LIN {X 112.363,Y 99.492,Z 63.257,A 180.000,B 0.000,C 180.000} C_DIS
LIN {X 112.396,Y 99.258,Z 63.249,A 180.000,B 0.000,C 180.000} C_DIS
LIN {X 112.406,Y 99.180,Z 63.246,A 180.000,B 0.000,C 180.000} C_DIS
LIN {X 112.413,Y 99.101,Z 63.243,A 180.000,B 0.000,C 180.000} C_DIS
LIN {X 112.420,Y 99.023,Z 63.241,A 180.000,B 0.000,C 180.000} C_DIS
LIN {X 112.433,Y 98.866,Z 63.235,A 180.000,B 0.000,C 180.000} C_DIS
LIN {X 112.453,Y 98.631,Z 63.227,A 180.000,B 0.000,C 180.000} C_DIS
LIN {X 112.466,Y 98.474,Z 63.221,A 180.000,B 0.000,C 180.000} C_DIS
LIN {X 112.473,Y 98.395,Z 63.219,A 180.000,B 0.000,C 180.000} C_DIS
LIN {X 112.478,Y 98.317,Z 63.216,A 180.000,B 0.000,C 180.000} C_DIS
LIN {X 112.480,Y 98.238,Z 63.213,A 180.000,B 0.000,C 180.000} C_DIS
LIN {X 112.494,Y 97.766,Z 63.197,A 180.000,B 0.000,C 180.000} C_DIS
LIN {X 112.498,Y 97.608,Z 63.191,A 180.000,B 0.000,C 180.000} C_DIS
LIN {X 112.500,Y 97.529,Z 63.188,A 180.000,B 0.000,C 180.000} C_DIS
LIN {X 112.500,Y 97.451,Z 63.186,A 180.000,B 0.000,C 180.000} C_DIS
LIN {X 112.497,Y 97.372,Z 63.183,A 180.000,B 0.000,C 180.000} C_DIS
LIN {X 112.493,Y 97.214,Z 63.177,A 180.000,B 0.000,C 180.000} C_DIS
LIN {X 112.491,Y 97.136,Z 63.175,A 180.000,B 0.000,C 180.000} C_DIS
LIN {X 112.486,Y 96.978,Z 63.169,A 180.000,B 0.000,C 180.000} C_DIS
LIN {X 112.480,Y 96.742,Z 63.161,A 180.000,B 0.000,C 180.000} C_DIS
LIN {X 112.477,Y 96.663,Z 63.158,A 180.000,B 0.000,C 180.000} C_DIS
LIN {X 112.471,Y 96.585,Z 63.155,A 180.000,B 0.000,C 180.000} C_DIS
LIN {X 112.458,Y 96.428,Z 63.150,A 180.000,B 0.000,C 180.000} C_DIS
LIN {X 112.418,Y 95.957,Z 63.133,A 180.000,B 0.000,C 180.000} C_DIS
LIN {X 112.412,Y 95.879,Z 63.131,A 180.000,B 0.000,C 180.000} C_DIS
LIN {X 112.403,Y 95.800,Z 63.128,A 180.000,B 0.000,C 180.000} C_DIS
LIN {X 112.393,Y 95.722,Z 63.125,A 180.000,B 0.000,C 180.000} C_DIS
LIN {X 112.305,Y 95.098,Z 63.103,A 180.000,B 0.000,C 180.000} C_DIS
LIN {X 112.293,Y 95.020,Z 63.100,A 180.000,B 0.000,C 180.000} C_DIS
LIN {X 112.280,Y 94.943,Z 63.098,A 180.000,B 0.000,C 180.000} C_DIS
LIN {X 112.265,Y 94.866,Z 63.095,A 180.000,B 0.000,C 180.000} C_DIS
LIN {X 112.142,Y 94.248,Z 63.073,A 180.000,B 0.000,C 180.000} C_DIS
LIN {X 112.126,Y 94.171,Z 63.070,A 180.000,B 0.000,C 180.000} C_DIS
LIN {X 112.107,Y 94.094,Z 63.067,A 180.000,B 0.000,C 180.000} C_DIS
LIN {X 111.989,Y 93.637,Z 63.051,A 180.000,B 0.000,C 180.000} C_DIS
LIN {X 111.930,Y 93.408,Z 63.043,A 180.000,B 0.000,C 180.000} C_DIS
LIN {X 111.909,Y 93.332,Z 63.040,A 180.000,B 0.000,C 180.000} C_DIS
LIN {X 111.886,Y 93.257,Z 63.037,A 180.000,B 0.000,C 180.000} C_DIS
LIN {X 111.695,Y 92.656,Z 63.015,A 180.000,B 0.000,C 180.000} C_DIS
LIN {X 111.670,Y 92.581,Z 63.012,A 180.000,B 0.000,C 180.000} C_DIS
LIN {X 111.644,Y 92.507,Z 63.010,A 180.000,B 0.000,C 180.000} C_DIS
LIN {X 111.616,Y 92.434,Z 63.007,A 180.000,B 0.000,C 180.000} C_DIS
LIN {X 111.392,Y 91.845,Z 62.985,A 180.000,B 0.000,C 180.000} C_DIS
LIN {X 111.363,Y 91.772,Z 62.982,A 180.000,B 0.000,C 180.000} C_DIS
LIN {X 111.332,Y 91.699,Z 62.979,A 180.000,B 0.000,C 180.000} C_DIS
LIN {X 111.203,Y 91.412,Z 62.968,A 180.000,B 0.000,C 180.000} C_DIS
LIN {X 111.043,Y 91.052,Z 62.955,A 180.000,B 0.000,C 180.000} C_DIS
LIN {X 111.009,Y 90.981,Z 62.952,A 180.000,B 0.000,C 180.000} C_DIS
LIN {X 110.974,Y 90.911,Z 62.949,A 180.000,B 0.000,C 180.000} C_DIS
LIN {X 110.685,Y 90.351,Z 62.927,A 180.000,B 0.000,C 180.000} C_DIS
LIN {X 110.648,Y 90.281,Z 62.924,A 180.000,B 0.000,C 180.000} C_DIS
LIN {X 110.610,Y 90.212,Z 62.922,A 180.000,B 0.000,C 180.000} C_DIS
LIN {X 110.570,Y 90.144,Z 62.919,A 180.000,B 0.000,C 180.000} C_DIS
LIN {X 110.250,Y 89.601,Z 62.897,A 180.000,B 0.000,C 180.000} C_DIS
LIN {X 110.210,Y 89.534,Z 62.894,A 180.000,B 0.000,C 180.000} C_DIS
LIN {X 110.167,Y 89.468,Z 62.891,A 180.000,B 0.000,C 180.000} C_DIS
LIN {X 110.124,Y 89.402,Z 62.889,A 180.000,B 0.000,C 180.000} C_DIS
LIN {X 109.992,Y 89.206,Z 62.880,A 180.000,B 0.000,C 180.000} C_DIS
LIN {X 109.905,Y 89.075,Z 62.875,A 180.000,B 0.000,C 180.000} C_DIS
LIN {X 109.774,Y 88.878,Z 62.867,A 180.000,B 0.000,C 180.000} C_DIS
LIN {X 109.729,Y 88.814,Z 62.864,A 180.000,B 0.000,C 180.000} C_DIS
LIN {X 109.682,Y 88.750,Z 62.861,A 180.000,B 0.000,C 180.000} C_DIS
LIN {X 109.351,Y 88.310,Z 62.842,A 180.000,B 0.000,C 180.000} C_DIS
LIN {X 109.303,Y 88.247,Z 62.839,A 180.000,B 0.000,C 180.000} C_DIS
LIN {X 109.256,Y 88.184,Z 62.836,A 180.000,B 0.000,C 180.000} C_DIS
LIN {X 109.207,Y 88.122,Z 62.834,A 180.000,B 0.000,C 180.000} C_DIS
LIN {X 109.156,Y 88.062,Z 62.831,A 180.000,B 0.000,C 180.000} C_DIS
LIN {X 109.055,Y 87.942,Z 62.825,A 180.000,B 0.000,C 180.000} C_DIS
LIN {X 109.004,Y 87.881,Z 62.823,A 180.000,B 0.000,C 180.000} C_DIS
LIN {X 108.902,Y 87.761,Z 62.817,A 180.000,B 0.000,C 180.000} C_DIS
LIN {X 108.750,Y 87.581,Z 62.809,A 180.000,B 0.000,C 180.000} C_DIS
LIN {X 108.699,Y 87.521,Z 62.806,A 180.000,B 0.000,C 180.000} C_DIS
LIN {X 108.646,Y 87.462,Z 62.803,A 180.000,B 0.000,C 180.000} C_DIS
LIN {X 108.592,Y 87.405,Z 62.801,A 180.000,B 0.000,C 180.000} C_DIS
LIN {X 108.483,Y 87.291,Z 62.795,A 180.000,B 0.000,C 180.000} C_DIS
LIN {X 108.159,Y 86.947,Z 62.779,A 180.000,B 0.000,C 180.000} C_DIS
LIN {X 108.104,Y 86.891,Z 62.776,A 180.000,B 0.000,C 180.000} C_DIS
LIN {X 108.047,Y 86.836,Z 62.773,A 180.000,B 0.000,C 180.000} C_DIS
LIN {X 107.876,Y 86.674,Z 62.765,A 180.000,B 0.000,C 180.000} C_DIS
LIN {X 107.761,Y 86.566,Z 62.759,A 180.000,B 0.000,C 180.000} C_DIS
LIN {X 107.704,Y 86.511,Z 62.757,A 180.000,B 0.000,C 180.000} C_DIS
LIN {X 107.590,Y 86.403,Z 62.751,A 180.000,B 0.000,C 180.000} C_DIS
LIN {X 107.532,Y 86.349,Z 62.748,A 180.000,B 0.000,C 180.000} C_DIS
LIN {X 107.474,Y 86.296,Z 62.746,A 180.000,B 0.000,C 180.000} C_DIS
LIN {X 107.414,Y 86.245,Z 62.743,A 180.000,B 0.000,C 180.000} C_DIS
LIN {X 107.294,Y 86.144,Z 62.737,A 180.000,B 0.000,C 180.000} C_DIS
LIN {X 107.233,Y 86.093,Z 62.735,A 180.000,B 0.000,C 180.000} C_DIS
LIN {X 107.113,Y 85.991,Z 62.729,A 180.000,B 0.000,C 180.000} C_DIS
LIN {X 106.933,Y 85.839,Z 62.721,A 180.000,B 0.000,C 180.000} C_DIS
LIN {X 106.872,Y 85.788,Z 62.718,A 180.000,B 0.000,C 180.000} C_DIS
LIN {X 106.810,Y 85.740,Z 62.715,A 180.000,B 0.000,C 180.000} C_DIS
LIN {X 106.747,Y 85.692,Z 62.713,A 180.000,B 0.000,C 180.000} C_DIS
LIN {X 106.622,Y 85.598,Z 62.707,A 180.000,B 0.000,C 180.000} C_DIS
LIN {X 106.433,Y 85.456,Z 62.699,A 180.000,B 0.000,C 180.000} C_DIS
LIN {X 106.307,Y 85.361,Z 62.693,A 180.000,B 0.000,C 180.000} C_DIS
LIN {X 106.244,Y 85.313,Z 62.691,A 180.000,B 0.000,C 180.000} C_DIS
LIN {X 106.180,Y 85.267,Z 62.688,A 180.000,B 0.000,C 180.000} C_DIS
LIN {X 106.116,Y 85.222,Z 62.685,A 180.000,B 0.000,C 180.000} C_DIS
LIN {X 105.985,Y 85.135,Z 62.680,A 180.000,B 0.000,C 180.000} C_DIS
LIN {X 105.854,Y 85.047,Z 62.674,A 180.000,B 0.000,C 180.000} C_DIS
LIN {X 105.723,Y 84.960,Z 62.669,A 180.000,B 0.000,C 180.000} C_DIS
LIN {X 105.592,Y 84.872,Z 62.664,A 180.000,B 0.000,C 180.000} C_DIS
LIN {X 105.526,Y 84.829,Z 62.661,A 180.000,B 0.000,C 180.000} C_DIS
LIN {X 105.460,Y 84.786,Z 62.659,A 180.000,B 0.000,C 180.000} C_DIS
LIN {X 105.392,Y 84.746,Z 62.656,A 180.000,B 0.000,C 180.000} C_DIS
LIN {X 105.324,Y 84.706,Z 62.654,A 180.000,B 0.000,C 180.000} C_DIS
LIN {X 105.257,Y 84.666,Z 62.651,A 180.000,B 0.000,C 180.000} C_DIS
LIN {X 105.189,Y 84.626,Z 62.649,A 180.000,B 0.000,C 180.000} C_DIS
LIN {X 105.053,Y 84.546,Z 62.644,A 180.000,B 0.000,C 180.000} C_DIS
LIN {X 104.917,Y 84.466,Z 62.639,A 180.000,B 0.000,C 180.000} C_DIS
LIN {X 104.782,Y 84.386,Z 62.634,A 180.000,B 0.000,C 180.000} C_DIS
LIN {X 104.643,Y 84.312,Z 62.629,A 180.000,B 0.000,C 180.000} C_DIS
LIN {X 104.503,Y 84.240,Z 62.624,A 180.000,B 0.000,C 180.000} C_DIS
LIN {X 104.363,Y 84.167,Z 62.620,A 180.000,B 0.000,C 180.000} C_DIS
LIN {X 104.223,Y 84.095,Z 62.615,A 180.000,B 0.000,C 180.000} C_DIS
LIN {X 104.083,Y 84.023,Z 62.610,A 180.000,B 0.000,C 180.000} C_DIS
LIN {X 103.941,Y 83.954,Z 62.606,A 180.000,B 0.000,C 180.000} C_DIS
LIN {X 103.797,Y 83.890,Z 62.602,A 180.000,B 0.000,C 180.000} C_DIS
LIN {X 103.654,Y 83.826,Z 62.597,A 180.000,B 0.000,C 180.000} C_DIS
LIN {X 103.510,Y 83.761,Z 62.593,A 180.000,B 0.000,C 180.000} C_DIS
LIN {X 103.366,Y 83.697,Z 62.589,A 180.000,B 0.000,C 180.000} C_DIS
LIN {X 103.222,Y 83.634,Z 62.585,A 180.000,B 0.000,C 180.000} C_DIS
LIN {X 103.075,Y 83.578,Z 62.581,A 180.000,B 0.000,C 180.000} C_DIS
LIN {X 102.927,Y 83.521,Z 62.577,A 180.000,B 0.000,C 180.000} C_DIS
LIN {X 102.780,Y 83.465,Z 62.573,A 180.000,B 0.000,C 180.000} C_DIS
LIN {X 102.633,Y 83.409,Z 62.570,A 180.000,B 0.000,C 180.000} C_DIS
LIN {X 102.486,Y 83.353,Z 62.566,A 180.000,B 0.000,C 180.000} C_DIS
LIN {X 102.337,Y 83.303,Z 62.562,A 180.000,B 0.000,C 180.000} C_DIS
LIN {X 102.186,Y 83.255,Z 62.559,A 180.000,B 0.000,C 180.000} C_DIS
LIN {X 102.036,Y 83.208,Z 62.556,A 180.000,B 0.000,C 180.000} C_DIS
LIN {X 101.886,Y 83.160,Z 62.552,A 180.000,B 0.000,C 180.000} C_DIS
LIN {X 101.736,Y 83.112,Z 62.549,A 180.000,B 0.000,C 180.000} C_DIS
LIN {X 101.585,Y 83.068,Z 62.546,A 180.000,B 0.000,C 180.000} C_DIS
LIN {X 101.433,Y 83.028,Z 62.543,A 180.000,B 0.000,C 180.000} C_DIS
LIN {X 101.280,Y 82.989,Z 62.540,A 180.000,B 0.000,C 180.000} C_DIS
LIN {X 101.128,Y 82.950,Z 62.537,A 180.000,B 0.000,C 180.000} C_DIS
LIN {X 100.975,Y 82.910,Z 62.534,A 180.000,B 0.000,C 180.000} C_DIS
LIN {X 100.822,Y 82.873,Z 62.532,A 180.000,B 0.000,C 180.000} C_DIS
LIN {X 100.668,Y 82.841,Z 62.529,A 180.000,B 0.000,C 180.000} C_DIS
LIN {X 100.513,Y 82.811,Z 62.527,A 180.000,B 0.000,C 180.000} C_DIS
LIN {X 100.204,Y 82.749,Z 62.522,A 180.000,B 0.000,C 180.000} C_DIS
LIN {X 99.894,Y 82.694,Z 62.518,A 180.000,B 0.000,C 180.000} C_DIS
LIN {X 99.582,Y 82.650,Z 62.514,A 180.000,B 0.000,C 180.000} C_DIS
LIN {X 99.270,Y 82.606,Z 62.511,A 180.000,B 0.000,C 180.000} C_DIS
LIN {X 98.957,Y 82.575,Z 62.508,A 180.000,B 0.000,C 180.000} C_DIS
LIN {X 98.643,Y 82.548,Z 62.505,A 180.000,B 0.000,C 180.000} C_DIS
LIN {X 98.329,Y 82.523,Z 62.503,A 180.000,B 0.000,C 180.000} C_DIS
LIN {X 98.014,Y 82.513,Z 62.502,A 180.000,B 0.000,C 180.000} C_DIS
LIN {X 97.699,Y 82.505,Z 62.501,A 180.000,B 0.000,C 180.000} C_DIS
LIN {X 97.385,Y 82.502,Z 62.500,A 180.000,B 0.000,C 180.000} C_DIS
LIN {X 97.153,Y 82.509,Z 62.500,A 180.000,B 0.000,C 180.000} C_DIS
; Cutting Move Starts
LIN {X 96.897,Y 82.516,Z 62.500,A 180.000,B 0.000,C 180.000} C_DIS
LIN {X 96.718,Y 82.521,Z 62.500,A 180.000,B 0.000,C 180.000} C_DIS
LIN {X 96.539,Y 82.533,Z 62.500,A 180.000,B 0.000,C 180.000} C_DIS
LIN {X 96.003,Y 82.578,Z 62.500,A 180.000,B 0.000,C 180.000} C_DIS
LIN {X 95.824,Y 82.594,Z 62.500,A 180.000,B 0.000,C 180.000} C_DIS
LIN {X 95.815,Y 82.595,Z 62.500,A 180.000,B 0.000,C 180.000} C_DIS
LIN {X 95.645,Y 82.618,Z 62.500,A 180.000,B 0.000,C 180.000} C_DIS
LIN {X 95.109,Y 82.694,Z 62.500,A 180.000,B 0.000,C 180.000} C_DIS
LIN {X 94.930,Y 82.722,Z 62.500,A 180.000,B 0.000,C 180.000} C_DIS
LIN {X 94.751,Y 82.758,Z 62.500,A 180.000,B 0.000,C 180.000} C_DIS
LIN {X 94.394,Y 82.829,Z 62.500,A 180.000,B 0.000,C 180.000} C_DIS
LIN {X 94.215,Y 82.865,Z 62.500,A 180.000,B 0.000,C 180.000} C_DIS
LIN {X 94.036,Y 82.908,Z 62.500,A 180.000,B 0.000,C 180.000} C_DIS
LIN {X 93.500,Y 83.046,Z 62.500,A 180.000,B 0.000,C 180.000} C_DIS
LIN {X 93.321,Y 83.094,Z 62.500,A 180.000,B 0.000,C 180.000} C_DIS
LIN {X 93.203,Y 83.131,Z 62.500,A 180.000,B 0.000,C 180.000} C_DIS
LIN {X 92.642,Y 83.310,Z 62.500,A 180.000,B 0.000,C 180.000} C_DIS
LIN {X 92.606,Y 83.322,Z 62.500,A 180.000,B 0.000,C 180.000} C_DIS
LIN {X 92.427,Y 83.386,Z 62.500,A 180.000,B 0.000,C 180.000} C_DIS
LIN {X 91.891,Y 83.591,Z 62.500,A 180.000,B 0.000,C 180.000} C_DIS
LIN {X 91.712,Y 83.662,Z 62.500,A 180.000,B 0.000,C 180.000} C_DIS
LIN {X 91.700,Y 83.668,Z 62.500,A 180.000,B 0.000,C 180.000} C_DIS
LIN {X 91.176,Y 83.902,Z 62.500,A 180.000,B 0.000,C 180.000} C_DIS
LIN {X 90.997,Y 83.983,Z 62.500,A 180.000,B 0.000,C 180.000} C_DIS
LIN {X 90.913,Y 84.025,Z 62.500,A 180.000,B 0.000,C 180.000} C_DIS
LIN {X 90.461,Y 84.259,Z 62.500,A 180.000,B 0.000,C 180.000} C_DIS
LIN {X 90.282,Y 84.351,Z 62.500,A 180.000,B 0.000,C 180.000} C_DIS
LIN {X 90.225,Y 84.383,Z 62.500,A 180.000,B 0.000,C 180.000} C_DIS
LIN {X 90.103,Y 84.454,Z 62.500,A 180.000,B 0.000,C 180.000} C_DIS
LIN {X 89.618,Y 84.740,Z 62.500,A 180.000,B 0.000,C 180.000} C_DIS
LIN {X 89.567,Y 84.770,Z 62.500,A 180.000,B 0.000,C 180.000} C_DIS
LIN {X 89.388,Y 84.886,Z 62.500,A 180.000,B 0.000,C 180.000} C_DIS
LIN {X 89.031,Y 85.125,Z 62.500,A 180.000,B 0.000,C 180.000} C_DIS
LIN {X 88.852,Y 85.244,Z 62.500,A 180.000,B 0.000,C 180.000} C_DIS
LIN {X 88.806,Y 85.276,Z 62.500,A 180.000,B 0.000,C 180.000} C_DIS
LIN {X 88.673,Y 85.376,Z 62.500,A 180.000,B 0.000,C 180.000} C_DIS
LIN {X 88.316,Y 85.645,Z 62.500,A 180.000,B 0.000,C 180.000} C_DIS
LIN {X 88.137,Y 85.781,Z 62.500,A 180.000,B 0.000,C 180.000} C_DIS
LIN {X 88.098,Y 85.813,Z 62.500,A 180.000,B 0.000,C 180.000} C_DIS
LIN {X 87.779,Y 86.082,Z 62.500,A 180.000,B 0.000,C 180.000} C_DIS
LIN {X 87.601,Y 86.233,Z 62.500,A 180.000,B 0.000,C 180.000} C_DIS
LIN {X 87.468,Y 86.349,Z 62.500,A 180.000,B 0.000,C 180.000} C_DIS
LIN {X 87.422,Y 86.393,Z 62.500,A 180.000,B 0.000,C 180.000} C_DIS
LIN {X 87.064,Y 86.731,Z 62.500,A 180.000,B 0.000,C 180.000} C_DIS
LIN {X 86.901,Y 86.885,Z 62.500,A 180.000,B 0.000,C 180.000} C_DIS
LIN {X 86.885,Y 86.901,Z 62.500,A 180.000,B 0.000,C 180.000} C_DIS
LIN {X 86.731,Y 87.064,Z 62.500,A 180.000,B 0.000,C 180.000} C_DIS
LIN {X 86.393,Y 87.422,Z 62.500,A 180.000,B 0.000,C 180.000} C_DIS
LIN {X 86.349,Y 87.468,Z 62.500,A 180.000,B 0.000,C 180.000} C_DIS
LIN {X 86.233,Y 87.601,Z 62.500,A 180.000,B 0.000,C 180.000} C_DIS
LIN {X 85.931,Y 87.958,Z 62.500,A 180.000,B 0.000,C 180.000} C_DIS
LIN {X 85.813,Y 88.098,Z 62.500,A 180.000,B 0.000,C 180.000} C_DIS
LIN {X 85.781,Y 88.137,Z 62.500,A 180.000,B 0.000,C 180.000} C_DIS
LIN {X 85.645,Y 88.316,Z 62.500,A 180.000,B 0.000,C 180.000} C_DIS
LIN {X 85.376,Y 88.673,Z 62.500,A 180.000,B 0.000,C 180.000} C_DIS
LIN {X 85.276,Y 88.806,Z 62.500,A 180.000,B 0.000,C 180.000} C_DIS
LIN {X 85.244,Y 88.852,Z 62.500,A 180.000,B 0.000,C 180.000} C_DIS
LIN {X 85.125,Y 89.031,Z 62.500,A 180.000,B 0.000,C 180.000} C_DIS
LIN {X 84.886,Y 89.388,Z 62.500,A 180.000,B 0.000,C 180.000} C_DIS
LIN {X 84.770,Y 89.567,Z 62.500,A 180.000,B 0.000,C 180.000} C_DIS
LIN {X 84.740,Y 89.618,Z 62.500,A 180.000,B 0.000,C 180.000} C_DIS
LIN {X 84.454,Y 90.103,Z 62.500,A 180.000,B 0.000,C 180.000} C_DIS
LIN {X 84.383,Y 90.225,Z 62.500,A 180.000,B 0.000,C 180.000} C_DIS
LIN {X 84.351,Y 90.282,Z 62.500,A 180.000,B 0.000,C 180.000} C_DIS
LIN {X 84.259,Y 90.461,Z 62.500,A 180.000,B 0.000,C 180.000} C_DIS
LIN {X 84.025,Y 90.913,Z 62.500,A 180.000,B 0.000,C 180.000} C_DIS
LIN {X 83.983,Y 90.997,Z 62.500,A 180.000,B 0.000,C 180.000} C_DIS
LIN {X 83.902,Y 91.176,Z 62.500,A 180.000,B 0.000,C 180.000} C_DIS
LIN {X 83.668,Y 91.700,Z 62.500,A 180.000,B 0.000,C 180.000} C_DIS
LIN {X 83.662,Y 91.712,Z 62.500,A 180.000,B 0.000,C 180.000} C_DIS
LIN {X 83.591,Y 91.891,Z 62.500,A 180.000,B 0.000,C 180.000} C_DIS
LIN {X 83.386,Y 92.427,Z 62.500,A 180.000,B 0.000,C 180.000} C_DIS
LIN {X 83.322,Y 92.606,Z 62.500,A 180.000,B 0.000,C 180.000} C_DIS
LIN {X 83.310,Y 92.642,Z 62.500,A 180.000,B 0.000,C 180.000} C_DIS
LIN {X 83.131,Y 93.203,Z 62.500,A 180.000,B 0.000,C 180.000} C_DIS
LIN {X 83.094,Y 93.321,Z 62.500,A 180.000,B 0.000,C 180.000} C_DIS
LIN {X 83.046,Y 93.500,Z 62.500,A 180.000,B 0.000,C 180.000} C_DIS
LIN {X 82.908,Y 94.036,Z 62.500,A 180.000,B 0.000,C 180.000} C_DIS
LIN {X 82.865,Y 94.215,Z 62.500,A 180.000,B 0.000,C 180.000} C_DIS
LIN {X 82.829,Y 94.394,Z 62.500,A 180.000,B 0.000,C 180.000} C_DIS
LIN {X 82.758,Y 94.751,Z 62.500,A 180.000,B 0.000,C 180.000} C_DIS
LIN {X 82.722,Y 94.930,Z 62.500,A 180.000,B 0.000,C 180.000} C_DIS
LIN {X 82.694,Y 95.109,Z 62.500,A 180.000,B 0.000,C 180.000} C_DIS
LIN {X 82.618,Y 95.645,Z 62.500,A 180.000,B 0.000,C 180.000} C_DIS
LIN {X 82.595,Y 95.815,Z 62.500,A 180.000,B 0.000,C 180.000} C_DIS
LIN {X 82.594,Y 95.824,Z 62.500,A 180.000,B 0.000,C 180.000} C_DIS
LIN {X 82.578,Y 96.003,Z 62.500,A 180.000,B 0.000,C 180.000} C_DIS
LIN {X 82.533,Y 96.539,Z 62.500,A 180.000,B 0.000,C 180.000} C_DIS
LIN {X 82.521,Y 96.718,Z 62.500,A 180.000,B 0.000,C 180.000} C_DIS
LIN {X 82.516,Y 96.897,Z 62.500,A 180.000,B 0.000,C 180.000} C_DIS
LIN {X 82.501,Y 97.433,Z 62.500,A 180.000,B 0.000,C 180.000} C_DIS
LIN {X 82.502,Y 97.612,Z 62.500,A 180.000,B 0.000,C 180.000} C_DIS
LIN {X 82.517,Y 98.148,Z 62.500,A 180.000,B 0.000,C 180.000} C_DIS
LIN {X 82.523,Y 98.327,Z 62.500,A 180.000,B 0.000,C 180.000} C_DIS
LIN {X 82.536,Y 98.505,Z 62.500,A 180.000,B 0.000,C 180.000} C_DIS
LIN {X 82.582,Y 99.042,Z 62.500,A 180.000,B 0.000,C 180.000} C_DIS
LIN {X 82.595,Y 99.185,Z 62.500,A 180.000,B 0.000,C 180.000} C_DIS
LIN {X 82.599,Y 99.221,Z 62.500,A 180.000,B 0.000,C 180.000} C_DIS
LIN {X 82.624,Y 99.399,Z 62.500,A 180.000,B 0.000,C 180.000} C_DIS
LIN {X 82.700,Y 99.936,Z 62.500,A 180.000,B 0.000,C 180.000} C_DIS
LIN {X 82.731,Y 100.114,Z 62.500,A 180.000,B 0.000,C 180.000} C_DIS
LIN {X 82.838,Y 100.651,Z 62.500,A 180.000,B 0.000,C 180.000} C_DIS
LIN {X 82.874,Y 100.829,Z 62.500,A 180.000,B 0.000,C 180.000} C_DIS
LIN {X 82.919,Y 101.008,Z 62.500,A 180.000,B 0.000,C 180.000} C_DIS
LIN {X 83.057,Y 101.545,Z 62.500,A 180.000,B 0.000,C 180.000} C_DIS
LIN {X 83.108,Y 101.723,Z 62.500,A 180.000,B 0.000,C 180.000} C_DIS
LIN {X 83.310,Y 102.358,Z 62.500,A 180.000,B 0.000,C 180.000} C_DIS
LIN {X 83.336,Y 102.438,Z 62.500,A 180.000,B 0.000,C 180.000} C_DIS
LIN {X 83.403,Y 102.617,Z 62.500,A 180.000,B 0.000,C 180.000} C_DIS
LIN {X 83.608,Y 103.153,Z 62.500,A 180.000,B 0.000,C 180.000} C_DIS
LIN {X 83.668,Y 103.300,Z 62.500,A 180.000,B 0.000,C 180.000} C_DIS
LIN {X 83.922,Y 103.869,Z 62.500,A 180.000,B 0.000,C 180.000} C_DIS
LIN {X 84.005,Y 104.047,Z 62.500,A 180.000,B 0.000,C 180.000} C_DIS
LIN {X 84.025,Y 104.087,Z 62.500,A 180.000,B 0.000,C 180.000} C_DIS
LIN {X 84.282,Y 104.584,Z 62.500,A 180.000,B 0.000,C 180.000} C_DIS
LIN {X 84.375,Y 104.762,Z 62.500,A 180.000,B 0.000,C 180.000} C_DIS
LIN {X 84.383,Y 104.775,Z 62.500,A 180.000,B 0.000,C 180.000} C_DIS
LIN {X 84.480,Y 104.941,Z 62.500,A 180.000,B 0.000,C 180.000} C_DIS
LIN {X 84.740,Y 105.382,Z 62.500,A 180.000,B 0.000,C 180.000} C_DIS
LIN {X 84.797,Y 105.477,Z 62.500,A 180.000,B 0.000,C 180.000} C_DIS
LIN {X 84.915,Y 105.656,Z 62.500,A 180.000,B 0.000,C 180.000} C_DIS
LIN {X 85.154,Y 106.014,Z 62.500,A 180.000,B 0.000,C 180.000} C_DIS
LIN {X 85.276,Y 106.193,Z 62.500,A 180.000,B 0.000,C 180.000} C_DIS
LIN {X 85.276,Y 106.194,Z 62.500,A 180.000,B 0.000,C 180.000} C_DIS
LIN {X 85.409,Y 106.371,Z 62.500,A 180.000,B 0.000,C 180.000} C_DIS
LIN {X 85.678,Y 106.729,Z 62.500,A 180.000,B 0.000,C 180.000} C_DIS
LIN {X 85.813,Y 106.902,Z 62.500,A 180.000,B 0.000,C 180.000} C_DIS
LIN {X 85.818,Y 106.908,Z 62.500,A 180.000,B 0.000,C 180.000} C_DIS
LIN {X 86.271,Y 107.444,Z 62.500,A 180.000,B 0.000,C 180.000} C_DIS
LIN {X 86.349,Y 107.532,Z 62.500,A 180.000,B 0.000,C 180.000} C_DIS
LIN {X 86.435,Y 107.623,Z 62.500,A 180.000,B 0.000,C 180.000} C_DIS
LIN {X 86.773,Y 107.980,Z 62.500,A 180.000,B 0.000,C 180.000} C_DIS
LIN {X 86.885,Y 108.099,Z 62.500,A 180.000,B 0.000,C 180.000} C_DIS
LIN {X 86.947,Y 108.159,Z 62.500,A 180.000,B 0.000,C 180.000} C_DIS
LIN {X 87.422,Y 108.607,Z 62.500,A 180.000,B 0.000,C 180.000} C_DIS
LIN {X 87.517,Y 108.695,Z 62.500,A 180.000,B 0.000,C 180.000} C_DIS
LIN {X 87.601,Y 108.767,Z 62.500,A 180.000,B 0.000,C 180.000} C_DIS
LIN {X 87.958,Y 109.069,Z 62.500,A 180.000,B 0.000,C 180.000} C_DIS
LIN {X 88.137,Y 109.219,Z 62.500,A 180.000,B 0.000,C 180.000} C_DIS
LIN {X 88.153,Y 109.232,Z 62.500,A 180.000,B 0.000,C 180.000} C_DIS
LIN {X 88.316,Y 109.355,Z 62.500,A 180.000,B 0.000,C 180.000} C_DIS
LIN {X 88.673,Y 109.624,Z 62.500,A 180.000,B 0.000,C 180.000} C_DIS
LIN {X 88.852,Y 109.756,Z 62.500,A 180.000,B 0.000,C 180.000} C_DIS
LIN {X 88.870,Y 109.768,Z 62.500,A 180.000,B 0.000,C 180.000} C_DIS
LIN {X 89.031,Y 109.875,Z 62.500,A 180.000,B 0.000,C 180.000} C_DIS
LIN {X 89.405,Y 110.126,Z 62.500,A 180.000,B 0.000,C 180.000} C_DIS
LIN {X 89.567,Y 110.230,Z 62.500,A 180.000,B 0.000,C 180.000} C_DIS
LIN {X 89.693,Y 110.304,Z 62.500,A 180.000,B 0.000,C 180.000} C_DIS
LIN {X 90.103,Y 110.546,Z 62.500,A 180.000,B 0.000,C 180.000} C_DIS
LIN {X 90.282,Y 110.649,Z 62.500,A 180.000,B 0.000,C 180.000} C_DIS
LIN {X 90.307,Y 110.662,Z 62.500,A 180.000,B 0.000,C 180.000} C_DIS
LIN {X 90.818,Y 110.926,Z 62.500,A 180.000,B 0.000,C 180.000} C_DIS
LIN {X 90.997,Y 111.017,Z 62.500,A 180.000,B 0.000,C 180.000} C_DIS
LIN {X 91.002,Y 111.019,Z 62.500,A 180.000,B 0.000,C 180.000} C_DIS
LIN {X 91.176,Y 111.098,Z 62.500,A 180.000,B 0.000,C 180.000} C_DIS
LIN {X 91.533,Y 111.258,Z 62.500,A 180.000,B 0.000,C 180.000} C_DIS
LIN {X 91.712,Y 111.338,Z 62.500,A 180.000,B 0.000,C 180.000} C_DIS
LIN {X 91.806,Y 111.377,Z 62.500,A 180.000,B 0.000,C 180.000} C_DIS
LIN {X 91.891,Y 111.409,Z 62.500,A 180.000,B 0.000,C 180.000} C_DIS
LIN {X 92.427,Y 111.614,Z 62.500,A 180.000,B 0.000,C 180.000} C_DIS
LIN {X 92.606,Y 111.678,Z 62.500,A 180.000,B 0.000,C 180.000} C_DIS
LIN {X 92.964,Y 111.792,Z 62.500,A 180.000,B 0.000,C 180.000} C_DIS
LIN {X 93.142,Y 111.849,Z 62.500,A 180.000,B 0.000,C 180.000} C_DIS
LIN {X 93.321,Y 111.906,Z 62.500,A 180.000,B 0.000,C 180.000} C_DIS
LIN {X 93.346,Y 111.913,Z 62.500,A 180.000,B 0.000,C 180.000} C_DIS
LIN {X 93.500,Y 111.954,Z 62.500,A 180.000,B 0.000,C 180.000} C_DIS
LIN {X 94.036,Y 112.092,Z 62.500,A 180.000,B 0.000,C 180.000} C_DIS
LIN {X 94.215,Y 112.135,Z 62.500,A 180.000,B 0.000,C 180.000} C_DIS
LIN {X 94.394,Y 112.171,Z 62.500,A 180.000,B 0.000,C 180.000} C_DIS
LIN {X 94.895,Y 112.271,Z 62.500,A 180.000,B 0.000,C 180.000} C_DIS
LIN {X 94.930,Y 112.278,Z 62.500,A 180.000,B 0.000,C 180.000} C_DIS
LIN {X 95.109,Y 112.306,Z 62.500,A 180.000,B 0.000,C 180.000} C_DIS
LIN {X 95.645,Y 112.382,Z 62.500,A 180.000,B 0.000,C 180.000} C_DIS
LIN {X 95.824,Y 112.406,Z 62.500,A 180.000,B 0.000,C 180.000} C_DIS
LIN {X 96.003,Y 112.422,Z 62.500,A 180.000,B 0.000,C 180.000} C_DIS
LIN {X 96.539,Y 112.467,Z 62.500,A 180.000,B 0.000,C 180.000} C_DIS
LIN {X 96.718,Y 112.479,Z 62.500,A 180.000,B 0.000,C 180.000} C_DIS
LIN {X 96.897,Y 112.484,Z 62.500,A 180.000,B 0.000,C 180.000} C_DIS
LIN {X 97.433,Y 112.499,Z 62.500,A 180.000,B 0.000,C 180.000} C_DIS
LIN {X 97.612,Y 112.498,Z 62.500,A 180.000,B 0.000,C 180.000} C_DIS
LIN {X 98.148,Y 112.483,Z 62.500,A 180.000,B 0.000,C 180.000} C_DIS
LIN {X 98.327,Y 112.477,Z 62.500,A 180.000,B 0.000,C 180.000} C_DIS
LIN {X 98.505,Y 112.464,Z 62.500,A 180.000,B 0.000,C 180.000} C_DIS
LIN {X 99.042,Y 112.418,Z 62.500,A 180.000,B 0.000,C 180.000} C_DIS
LIN {X 99.221,Y 112.401,Z 62.500,A 180.000,B 0.000,C 180.000} C_DIS
LIN {X 99.399,Y 112.376,Z 62.500,A 180.000,B 0.000,C 180.000} C_DIS
LIN {X 99.936,Y 112.300,Z 62.500,A 180.000,B 0.000,C 180.000} C_DIS
LIN {X 100.105,Y 112.271,Z 62.500,A 180.000,B 0.000,C 180.000} C_DIS
LIN {X 100.651,Y 112.162,Z 62.500,A 180.000,B 0.000,C 180.000} C_DIS
LIN {X 100.829,Y 112.126,Z 62.500,A 180.000,B 0.000,C 180.000} C_DIS
LIN {X 100.966,Y 112.092,Z 62.500,A 180.000,B 0.000,C 180.000} C_DIS
LIN {X 101.545,Y 111.943,Z 62.500,A 180.000,B 0.000,C 180.000} C_DIS
LIN {X 101.654,Y 111.913,Z 62.500,A 180.000,B 0.000,C 180.000} C_DIS
LIN {X 101.723,Y 111.892,Z 62.500,A 180.000,B 0.000,C 180.000} C_DIS
LIN {X 102.260,Y 111.721,Z 62.500,A 180.000,B 0.000,C 180.000} C_DIS
LIN {X 102.438,Y 111.664,Z 62.500,A 180.000,B 0.000,C 180.000} C_DIS
LIN {X 102.617,Y 111.597,Z 62.500,A 180.000,B 0.000,C 180.000} C_DIS
LIN {X 103.153,Y 111.392,Z 62.500,A 180.000,B 0.000,C 180.000} C_DIS
LIN {X 103.194,Y 111.377,Z 62.500,A 180.000,B 0.000,C 180.000} C_DIS
LIN {X 103.332,Y 111.318,Z 62.500,A 180.000,B 0.000,C 180.000} C_DIS
LIN {X 103.869,Y 111.078,Z 62.500,A 180.000,B 0.000,C 180.000} C_DIS
LIN {X 103.998,Y 111.019,Z 62.500,A 180.000,B 0.000,C 180.000} C_DIS
LIN {X 104.047,Y 110.995,Z 62.500,A 180.000,B 0.000,C 180.000} C_DIS
LIN {X 104.226,Y 110.903,Z 62.500,A 180.000,B 0.000,C 180.000} C_DIS
LIN {X 104.693,Y 110.662,Z 62.500,A 180.000,B 0.000,C 180.000} C_DIS
LIN {X 104.762,Y 110.625,Z 62.500,A 180.000,B 0.000,C 180.000} C_DIS
LIN {X 104.941,Y 110.520,Z 62.500,A 180.000,B 0.000,C 180.000} C_DIS
LIN {X 105.307,Y 110.304,Z 62.500,A 180.000,B 0.000,C 180.000} C_DIS
LIN {X 105.477,Y 110.203,Z 62.500,A 180.000,B 0.000,C 180.000} C_DIS
LIN {X 105.595,Y 110.126,Z 62.500,A 180.000,B 0.000,C 180.000} C_DIS
LIN {X 106.014,Y 109.846,Z 62.500,A 180.000,B 0.000,C 180.000} C_DIS
LIN {X 106.130,Y 109.768,Z 62.500,A 180.000,B 0.000,C 180.000} C_DIS
LIN {X 106.193,Y 109.724,Z 62.500,A 180.000,B 0.000,C 180.000} C_DIS
LIN {X 106.371,Y 109.591,Z 62.500,A 180.000,B 0.000,C 180.000} C_DIS
LIN {X 106.729,Y 109.322,Z 62.500,A 180.000,B 0.000,C 180.000} C_DIS
LIN {X 106.847,Y 109.232,Z 62.500,A 180.000,B 0.000,C 180.000} C_DIS
LIN {X 106.908,Y 109.182,Z 62.500,A 180.000,B 0.000,C 180.000} C_DIS
LIN {X 107.444,Y 108.729,Z 62.500,A 180.000,B 0.000,C 180.000} C_DIS
LIN {X 107.483,Y 108.695,Z 62.500,A 180.000,B 0.000,C 180.000} C_DIS
LIN {X 107.623,Y 108.565,Z 62.500,A 180.000,B 0.000,C 180.000} C_DIS
LIN {X 108.053,Y 108.159,Z 62.500,A 180.000,B 0.000,C 180.000} C_DIS
LIN {X 108.159,Y 108.053,Z 62.500,A 180.000,B 0.000,C 180.000} C_DIS
LIN {X 108.565,Y 107.623,Z 62.500,A 180.000,B 0.000,C 180.000} C_DIS
LIN {X 108.695,Y 107.483,Z 62.500,A 180.000,B 0.000,C 180.000} C_DIS
LIN {X 108.729,Y 107.444,Z 62.500,A 180.000,B 0.000,C 180.000} C_DIS
LIN {X 109.182,Y 106.908,Z 62.500,A 180.000,B 0.000,C 180.000} C_DIS
LIN {X 109.232,Y 106.847,Z 62.500,A 180.000,B 0.000,C 180.000} C_DIS
LIN {X 109.322,Y 106.729,Z 62.500,A 180.000,B 0.000,C 180.000} C_DIS
LIN {X 109.591,Y 106.371,Z 62.500,A 180.000,B 0.000,C 180.000} C_DIS
LIN {X 109.724,Y 106.193,Z 62.500,A 180.000,B 0.000,C 180.000} C_DIS
LIN {X 109.768,Y 106.130,Z 62.500,A 180.000,B 0.000,C 180.000} C_DIS
LIN {X 109.846,Y 106.014,Z 62.500,A 180.000,B 0.000,C 180.000} C_DIS
LIN {X 110.126,Y 105.595,Z 62.500,A 180.000,B 0.000,C 180.000} C_DIS
LIN {X 110.203,Y 105.477,Z 62.500,A 180.000,B 0.000,C 180.000} C_DIS
LIN {X 110.304,Y 105.307,Z 62.500,A 180.000,B 0.000,C 180.000} C_DIS
LIN {X 110.520,Y 104.941,Z 62.500,A 180.000,B 0.000,C 180.000} C_DIS
LIN {X 110.625,Y 104.762,Z 62.500,A 180.000,B 0.000,C 180.000} C_DIS
LIN {X 110.662,Y 104.693,Z 62.500,A 180.000,B 0.000,C 180.000} C_DIS
LIN {X 110.903,Y 104.226,Z 62.500,A 180.000,B 0.000,C 180.000} C_DIS
LIN {X 110.995,Y 104.047,Z 62.500,A 180.000,B 0.000,C 180.000} C_DIS
LIN {X 111.019,Y 103.998,Z 62.500,A 180.000,B 0.000,C 180.000} C_DIS
LIN {X 111.078,Y 103.869,Z 62.500,A 180.000,B 0.000,C 180.000} C_DIS
LIN {X 111.318,Y 103.332,Z 62.500,A 180.000,B 0.000,C 180.000} C_DIS
LIN {X 111.377,Y 103.194,Z 62.500,A 180.000,B 0.000,C 180.000} C_DIS
LIN {X 111.392,Y 103.153,Z 62.500,A 180.000,B 0.000,C 180.000} C_DIS
LIN {X 111.597,Y 102.617,Z 62.500,A 180.000,B 0.000,C 180.000} C_DIS
LIN {X 111.664,Y 102.438,Z 62.500,A 180.000,B 0.000,C 180.000} C_DIS
LIN {X 111.721,Y 102.260,Z 62.500,A 180.000,B 0.000,C 180.000} C_DIS
LIN {X 111.892,Y 101.723,Z 62.500,A 180.000,B 0.000,C 180.000} C_DIS
LIN {X 111.913,Y 101.654,Z 62.500,A 180.000,B 0.000,C 180.000} C_DIS
LIN {X 111.943,Y 101.545,Z 62.500,A 180.000,B 0.000,C 180.000} C_DIS
LIN {X 112.092,Y 100.966,Z 62.500,A 180.000,B 0.000,C 180.000} C_DIS
LIN {X 112.126,Y 100.829,Z 62.500,A 180.000,B 0.000,C 180.000} C_DIS
LIN {X 112.162,Y 100.651,Z 62.500,A 180.000,B 0.000,C 180.000} C_DIS
LIN {X 112.271,Y 100.105,Z 62.500,A 180.000,B 0.000,C 180.000} C_DIS
LIN {X 112.300,Y 99.936,Z 62.500,A 180.000,B 0.000,C 180.000} C_DIS
LIN {X 112.376,Y 99.399,Z 62.500,A 180.000,B 0.000,C 180.000} C_DIS
LIN {X 112.401,Y 99.221,Z 62.500,A 180.000,B 0.000,C 180.000} C_DIS
LIN {X 112.418,Y 99.042,Z 62.500,A 180.000,B 0.000,C 180.000} C_DIS
LIN {X 112.464,Y 98.505,Z 62.500,A 180.000,B 0.000,C 180.000} C_DIS
LIN {X 112.477,Y 98.327,Z 62.500,A 180.000,B 0.000,C 180.000} C_DIS
LIN {X 112.483,Y 98.148,Z 62.500,A 180.000,B 0.000,C 180.000} C_DIS
LIN {X 112.498,Y 97.612,Z 62.500,A 180.000,B 0.000,C 180.000} C_DIS
LIN {X 112.499,Y 97.433,Z 62.500,A 180.000,B 0.000,C 180.000} C_DIS
LIN {X 112.484,Y 96.897,Z 62.500,A 180.000,B 0.000,C 180.000} C_DIS
LIN {X 112.479,Y 96.718,Z 62.500,A 180.000,B 0.000,C 180.000} C_DIS
LIN {X 112.467,Y 96.539,Z 62.500,A 180.000,B 0.000,C 180.000} C_DIS
LIN {X 112.422,Y 96.003,Z 62.500,A 180.000,B 0.000,C 180.000} C_DIS
LIN {X 112.406,Y 95.824,Z 62.500,A 180.000,B 0.000,C 180.000} C_DIS
LIN {X 112.382,Y 95.645,Z 62.500,A 180.000,B 0.000,C 180.000} C_DIS
LIN {X 112.306,Y 95.109,Z 62.500,A 180.000,B 0.000,C 180.000} C_DIS
LIN {X 112.278,Y 94.930,Z 62.500,A 180.000,B 0.000,C 180.000} C_DIS
LIN {X 112.271,Y 94.895,Z 62.500,A 180.000,B 0.000,C 180.000} C_DIS
LIN {X 112.171,Y 94.394,Z 62.500,A 180.000,B 0.000,C 180.000} C_DIS
LIN {X 112.135,Y 94.215,Z 62.500,A 180.000,B 0.000,C 180.000} C_DIS
LIN {X 112.092,Y 94.036,Z 62.500,A 180.000,B 0.000,C 180.000} C_DIS
LIN {X 111.954,Y 93.500,Z 62.500,A 180.000,B 0.000,C 180.000} C_DIS
LIN {X 111.913,Y 93.346,Z 62.500,A 180.000,B 0.000,C 180.000} C_DIS
LIN {X 111.906,Y 93.321,Z 62.500,A 180.000,B 0.000,C 180.000} C_DIS
LIN {X 111.849,Y 93.142,Z 62.500,A 180.000,B 0.000,C 180.000} C_DIS
LIN {X 111.734,Y 92.782,Z 62.500,A 180.000,B 0.000,C 180.000} C_DIS
LIN {X 111.678,Y 92.606,Z 62.500,A 180.000,B 0.000,C 180.000} C_DIS
LIN {X 111.614,Y 92.427,Z 62.500,A 180.000,B 0.000,C 180.000} C_DIS
LIN {X 111.409,Y 91.891,Z 62.500,A 180.000,B 0.000,C 180.000} C_DIS
LIN {X 111.377,Y 91.806,Z 62.500,A 180.000,B 0.000,C 180.000} C_DIS
LIN {X 111.338,Y 91.712,Z 62.500,A 180.000,B 0.000,C 180.000} C_DIS
LIN {X 111.258,Y 91.533,Z 62.500,A 180.000,B 0.000,C 180.000} C_DIS
LIN {X 111.098,Y 91.176,Z 62.500,A 180.000,B 0.000,C 180.000} C_DIS
LIN {X 111.019,Y 91.002,Z 62.500,A 180.000,B 0.000,C 180.000} C_DIS
LIN {X 111.017,Y 90.997,Z 62.500,A 180.000,B 0.000,C 180.000} C_DIS
LIN {X 110.926,Y 90.818,Z 62.500,A 180.000,B 0.000,C 180.000} C_DIS
LIN {X 110.662,Y 90.307,Z 62.500,A 180.000,B 0.000,C 180.000} C_DIS
LIN {X 110.649,Y 90.282,Z 62.500,A 180.000,B 0.000,C 180.000} C_DIS
LIN {X 110.546,Y 90.103,Z 62.500,A 180.000,B 0.000,C 180.000} C_DIS
LIN {X 110.304,Y 89.693,Z 62.500,A 180.000,B 0.000,C 180.000} C_DIS
LIN {X 110.230,Y 89.567,Z 62.500,A 180.000,B 0.000,C 180.000} C_DIS
LIN {X 110.126,Y 89.405,Z 62.500,A 180.000,B 0.000,C 180.000} C_DIS
LIN {X 109.875,Y 89.031,Z 62.500,A 180.000,B 0.000,C 180.000} C_DIS
LIN {X 109.768,Y 88.870,Z 62.500,A 180.000,B 0.000,C 180.000} C_DIS
LIN {X 109.756,Y 88.852,Z 62.500,A 180.000,B 0.000,C 180.000} C_DIS
LIN {X 109.624,Y 88.673,Z 62.500,A 180.000,B 0.000,C 180.000} C_DIS
LIN {X 109.355,Y 88.316,Z 62.500,A 180.000,B 0.000,C 180.000} C_DIS
LIN {X 109.232,Y 88.153,Z 62.500,A 180.000,B 0.000,C 180.000} C_DIS
LIN {X 109.219,Y 88.137,Z 62.500,A 180.000,B 0.000,C 180.000} C_DIS
LIN {X 109.069,Y 87.958,Z 62.500,A 180.000,B 0.000,C 180.000} C_DIS
LIN {X 108.767,Y 87.601,Z 62.500,A 180.000,B 0.000,C 180.000} C_DIS
LIN {X 108.695,Y 87.517,Z 62.500,A 180.000,B 0.000,C 180.000} C_DIS
LIN {X 108.607,Y 87.422,Z 62.500,A 180.000,B 0.000,C 180.000} C_DIS
LIN {X 108.159,Y 86.947,Z 62.500,A 180.000,B 0.000,C 180.000} C_DIS
LIN {X 108.099,Y 86.885,Z 62.500,A 180.000,B 0.000,C 180.000} C_DIS
LIN {X 107.980,Y 86.773,Z 62.500,A 180.000,B 0.000,C 180.000} C_DIS
LIN {X 107.623,Y 86.435,Z 62.500,A 180.000,B 0.000,C 180.000} C_DIS
LIN {X 107.532,Y 86.349,Z 62.500,A 180.000,B 0.000,C 180.000} C_DIS
LIN {X 107.444,Y 86.271,Z 62.500,A 180.000,B 0.000,C 180.000} C_DIS
LIN {X 106.908,Y 85.818,Z 62.500,A 180.000,B 0.000,C 180.000} C_DIS
LIN {X 106.902,Y 85.813,Z 62.500,A 180.000,B 0.000,C 180.000} C_DIS
LIN {X 106.729,Y 85.678,Z 62.500,A 180.000,B 0.000,C 180.000} C_DIS
LIN {X 106.371,Y 85.409,Z 62.500,A 180.000,B 0.000,C 180.000} C_DIS
LIN {X 106.194,Y 85.276,Z 62.500,A 180.000,B 0.000,C 180.000} C_DIS
LIN {X 106.193,Y 85.276,Z 62.500,A 180.000,B 0.000,C 180.000} C_DIS
LIN {X 106.014,Y 85.154,Z 62.500,A 180.000,B 0.000,C 180.000} C_DIS
LIN {X 105.656,Y 84.915,Z 62.500,A 180.000,B 0.000,C 180.000} C_DIS
LIN {X 105.477,Y 84.797,Z 62.500,A 180.000,B 0.000,C 180.000} C_DIS
LIN {X 105.382,Y 84.740,Z 62.500,A 180.000,B 0.000,C 180.000} C_DIS
LIN {X 104.941,Y 84.480,Z 62.500,A 180.000,B 0.000,C 180.000} C_DIS
LIN {X 104.775,Y 84.383,Z 62.500,A 180.000,B 0.000,C 180.000} C_DIS
LIN {X 104.762,Y 84.375,Z 62.500,A 180.000,B 0.000,C 180.000} C_DIS
LIN {X 104.584,Y 84.282,Z 62.500,A 180.000,B 0.000,C 180.000} C_DIS
LIN {X 104.087,Y 84.025,Z 62.500,A 180.000,B 0.000,C 180.000} C_DIS
LIN {X 104.047,Y 84.005,Z 62.500,A 180.000,B 0.000,C 180.000} C_DIS
LIN {X 103.869,Y 83.922,Z 62.500,A 180.000,B 0.000,C 180.000} C_DIS
LIN {X 103.300,Y 83.668,Z 62.500,A 180.000,B 0.000,C 180.000} C_DIS
LIN {X 103.153,Y 83.608,Z 62.500,A 180.000,B 0.000,C 180.000} C_DIS
LIN {X 102.617,Y 83.403,Z 62.500,A 180.000,B 0.000,C 180.000} C_DIS
LIN {X 102.438,Y 83.336,Z 62.500,A 180.000,B 0.000,C 180.000} C_DIS
LIN {X 102.358,Y 83.310,Z 62.500,A 180.000,B 0.000,C 180.000} C_DIS
LIN {X 101.723,Y 83.108,Z 62.500,A 180.000,B 0.000,C 180.000} C_DIS
LIN {X 101.545,Y 83.057,Z 62.500,A 180.000,B 0.000,C 180.000} C_DIS
LIN {X 101.008,Y 82.919,Z 62.500,A 180.000,B 0.000,C 180.000} C_DIS
LIN {X 100.829,Y 82.874,Z 62.500,A 180.000,B 0.000,C 180.000} C_DIS
LIN {X 100.651,Y 82.838,Z 62.500,A 180.000,B 0.000,C 180.000} C_DIS
LIN {X 100.114,Y 82.731,Z 62.500,A 180.000,B 0.000,C 180.000} C_DIS
LIN {X 99.936,Y 82.700,Z 62.500,A 180.000,B 0.000,C 180.000} C_DIS
LIN {X 99.399,Y 82.624,Z 62.500,A 180.000,B 0.000,C 180.000} C_DIS
LIN {X 99.221,Y 82.599,Z 62.500,A 180.000,B 0.000,C 180.000} C_DIS
LIN {X 99.185,Y 82.595,Z 62.500,A 180.000,B 0.000,C 180.000} C_DIS
LIN {X 99.042,Y 82.582,Z 62.500,A 180.000,B 0.000,C 180.000} C_DIS
LIN {X 98.505,Y 82.536,Z 62.500,A 180.000,B 0.000,C 180.000} C_DIS
LIN {X 98.327,Y 82.523,Z 62.500,A 180.000,B 0.000,C 180.000} C_DIS
LIN {X 98.148,Y 82.517,Z 62.500,A 180.000,B 0.000,C 180.000} C_DIS
LIN {X 97.612,Y 82.502,Z 62.500,A 180.000,B 0.000,C 180.000} C_DIS
LIN {X 97.433,Y 82.501,Z 62.500,A 180.000,B 0.000,C 180.000} C_DIS
LIN {X 97.153,Y 82.509,Z 62.500,A 180.000,B 0.000,C 180.000} C_DIS
; Link Move Starts
LIN {X 96.838,Y 82.518,Z 62.500,A 180.000,B 0.000,C 180.000} C_DIS
LIN {X 96.524,Y 82.534,Z 62.498,A 180.000,B 0.000,C 180.000} C_DIS
LIN {X 96.210,Y 82.561,Z 62.496,A 180.000,B 0.000,C 180.000} C_DIS
LIN {X 95.896,Y 82.587,Z 62.492,A 180.000,B 0.000,C 180.000} C_DIS
LIN {X 95.583,Y 82.627,Z 62.488,A 180.000,B 0.000,C 180.000} C_DIS
LIN {X 95.272,Y 82.671,Z 62.483,A 180.000,B 0.000,C 180.000} C_DIS
LIN {X 95.116,Y 82.693,Z 62.481,A 180.000,B 0.000,C 180.000} C_DIS
LIN {X 94.960,Y 82.717,Z 62.478,A 180.000,B 0.000,C 180.000} C_DIS
LIN {X 94.805,Y 82.747,Z 62.475,A 180.000,B 0.000,C 180.000} C_DIS
LIN {X 94.651,Y 82.778,Z 62.471,A 180.000,B 0.000,C 180.000} C_DIS
LIN {X 94.496,Y 82.809,Z 62.468,A 180.000,B 0.000,C 180.000} C_DIS
LIN {X 94.342,Y 82.839,Z 62.464,A 180.000,B 0.000,C 180.000} C_DIS
LIN {X 94.188,Y 82.870,Z 62.460,A 180.000,B 0.000,C 180.000} C_DIS
LIN {X 94.035,Y 82.908,Z 62.456,A 180.000,B 0.000,C 180.000} C_DIS
LIN {X 93.882,Y 82.947,Z 62.452,A 180.000,B 0.000,C 180.000} C_DIS
LIN {X 93.730,Y 82.987,Z 62.448,A 180.000,B 0.000,C 180.000} C_DIS
LIN {X 93.577,Y 83.026,Z 62.444,A 180.000,B 0.000,C 180.000} C_DIS
LIN {X 93.425,Y 83.065,Z 62.439,A 180.000,B 0.000,C 180.000} C_DIS
LIN {X 93.273,Y 83.109,Z 62.434,A 180.000,B 0.000,C 180.000} C_DIS
LIN {X 93.123,Y 83.157,Z 62.429,A 180.000,B 0.000,C 180.000} C_DIS
LIN {X 92.973,Y 83.205,Z 62.424,A 180.000,B 0.000,C 180.000} C_DIS
LIN {X 92.898,Y 83.228,Z 62.422,A 180.000,B 0.000,C 180.000} C_DIS
LIN {X 92.823,Y 83.252,Z 62.419,A 180.000,B 0.000,C 180.000} C_DIS
LIN {X 92.748,Y 83.276,Z 62.417,A 180.000,B 0.000,C 180.000} C_DIS
LIN {X 92.673,Y 83.300,Z 62.414,A 180.000,B 0.000,C 180.000} C_DIS
LIN {X 92.598,Y 83.324,Z 62.411,A 180.000,B 0.000,C 180.000} C_DIS
LIN {X 92.523,Y 83.350,Z 62.409,A 180.000,B 0.000,C 180.000} C_DIS
LIN {X 92.450,Y 83.377,Z 62.406,A 180.000,B 0.000,C 180.000} C_DIS
LIN {X 92.376,Y 83.405,Z 62.403,A 180.000,B 0.000,C 180.000} C_DIS
LIN {X 92.303,Y 83.434,Z 62.401,A 180.000,B 0.000,C 180.000} C_DIS
LIN {X 92.229,Y 83.462,Z 62.398,A 180.000,B 0.000,C 180.000} C_DIS
LIN {X 92.155,Y 83.490,Z 62.395,A 180.000,B 0.000,C 180.000} C_DIS
LIN {X 92.082,Y 83.518,Z 62.392,A 180.000,B 0.000,C 180.000} C_DIS
LIN {X 92.008,Y 83.546,Z 62.389,A 180.000,B 0.000,C 180.000} C_DIS
LIN {X 91.935,Y 83.574,Z 62.387,A 180.000,B 0.000,C 180.000} C_DIS
LIN {X 91.861,Y 83.602,Z 62.384,A 180.000,B 0.000,C 180.000} C_DIS
LIN {X 91.788,Y 83.630,Z 62.381,A 180.000,B 0.000,C 180.000} C_DIS
LIN {X 91.715,Y 83.661,Z 62.378,A 180.000,B 0.000,C 180.000} C_DIS
LIN {X 91.643,Y 83.693,Z 62.376,A 180.000,B 0.000,C 180.000} C_DIS
LIN {X 91.571,Y 83.725,Z 62.373,A 180.000,B 0.000,C 180.000} C_DIS
LIN {X 91.499,Y 83.757,Z 62.370,A 180.000,B 0.000,C 180.000} C_DIS
LIN {X 91.427,Y 83.789,Z 62.367,A 180.000,B 0.000,C 180.000} C_DIS
LIN {X 91.356,Y 83.822,Z 62.365,A 180.000,B 0.000,C 180.000} C_DIS
LIN {X 91.284,Y 83.854,Z 62.362,A 180.000,B 0.000,C 180.000} C_DIS
LIN {X 91.140,Y 83.918,Z 62.356,A 180.000,B 0.000,C 180.000} C_DIS
LIN {X 91.068,Y 83.950,Z 62.354,A 180.000,B 0.000,C 180.000} C_DIS
LIN {X 90.997,Y 83.983,Z 62.351,A 180.000,B 0.000,C 180.000} C_DIS
LIN {X 90.926,Y 84.018,Z 62.348,A 180.000,B 0.000,C 180.000} C_DIS
LIN {X 90.716,Y 84.127,Z 62.340,A 180.000,B 0.000,C 180.000} C_DIS
LIN {X 90.576,Y 84.199,Z 62.334,A 180.000,B 0.000,C 180.000} C_DIS
LIN {X 90.506,Y 84.235,Z 62.332,A 180.000,B 0.000,C 180.000} C_DIS
LIN {X 90.366,Y 84.307,Z 62.326,A 180.000,B 0.000,C 180.000} C_DIS
LIN {X 90.296,Y 84.344,Z 62.323,A 180.000,B 0.000,C 180.000} C_DIS
LIN {X 90.227,Y 84.381,Z 62.321,A 180.000,B 0.000,C 180.000} C_DIS
LIN {X 90.159,Y 84.421,Z 62.318,A 180.000,B 0.000,C 180.000} C_DIS
LIN {X 90.023,Y 84.501,Z 62.312,A 180.000,B 0.000,C 180.000} C_DIS
LIN {X 89.956,Y 84.541,Z 62.310,A 180.000,B 0.000,C 180.000} C_DIS
LIN {X 89.820,Y 84.621,Z 62.304,A 180.000,B 0.000,C 180.000} C_DIS
LIN {X 89.616,Y 84.741,Z 62.296,A 180.000,B 0.000,C 180.000} C_DIS
LIN {X 89.549,Y 84.781,Z 62.293,A 180.000,B 0.000,C 180.000} C_DIS
LIN {X 89.482,Y 84.823,Z 62.290,A 180.000,B 0.000,C 180.000} C_DIS
LIN {X 89.417,Y 84.867,Z 62.288,A 180.000,B 0.000,C 180.000} C_DIS
LIN {X 89.220,Y 84.998,Z 62.279,A 180.000,B 0.000,C 180.000} C_DIS
LIN {X 89.089,Y 85.086,Z 62.274,A 180.000,B 0.000,C 180.000} C_DIS
LIN {X 88.893,Y 85.217,Z 62.266,A 180.000,B 0.000,C 180.000} C_DIS
LIN {X 88.828,Y 85.261,Z 62.263,A 180.000,B 0.000,C 180.000} C_DIS
LIN {X 88.764,Y 85.307,Z 62.260,A 180.000,B 0.000,C 180.000} C_DIS
LIN {X 88.198,Y 85.734,Z 62.235,A 180.000,B 0.000,C 180.000} C_DIS
LIN {X 88.136,Y 85.782,Z 62.233,A 180.000,B 0.000,C 180.000} C_DIS
LIN {X 88.075,Y 85.832,Z 62.230,A 180.000,B 0.000,C 180.000} C_DIS
LIN {X 87.594,Y 86.239,Z 62.208,A 180.000,B 0.000,C 180.000} C_DIS
LIN {X 87.534,Y 86.290,Z 62.205,A 180.000,B 0.000,C 180.000} C_DIS
LIN {X 87.475,Y 86.342,Z 62.202,A 180.000,B 0.000,C 180.000} C_DIS
LIN {X 87.418,Y 86.396,Z 62.200,A 180.000,B 0.000,C 180.000} C_DIS
LIN {X 87.303,Y 86.505,Z 62.194,A 180.000,B 0.000,C 180.000} C_DIS
LIN {X 86.960,Y 86.829,Z 62.178,A 180.000,B 0.000,C 180.000} C_DIS
LIN {X 86.903,Y 86.884,Z 62.175,A 180.000,B 0.000,C 180.000} C_DIS
LIN {X 86.848,Y 86.940,Z 62.172,A 180.000,B 0.000,C 180.000} C_DIS
LIN {X 86.740,Y 87.054,Z 62.167,A 180.000,B 0.000,C 180.000} C_DIS
LIN {X 86.632,Y 87.169,Z 62.161,A 180.000,B 0.000,C 180.000} C_DIS
LIN {X 86.469,Y 87.341,Z 62.153,A 180.000,B 0.000,C 180.000} C_DIS
LIN {X 86.361,Y 87.455,Z 62.147,A 180.000,B 0.000,C 180.000} C_DIS
LIN {X 86.308,Y 87.513,Z 62.145,A 180.000,B 0.000,C 180.000} C_DIS
LIN {X 86.257,Y 87.573,Z 62.142,A 180.000,B 0.000,C 180.000} C_DIS
LIN {X 86.155,Y 87.693,Z 62.136,A 180.000,B 0.000,C 180.000} C_DIS
LIN {X 86.104,Y 87.753,Z 62.134,A 180.000,B 0.000,C 180.000} C_DIS
LIN {X 86.053,Y 87.814,Z 62.131,A 180.000,B 0.000,C 180.000} C_DIS
LIN {X 86.003,Y 87.874,Z 62.128,A 180.000,B 0.000,C 180.000} C_DIS
LIN {X 85.952,Y 87.934,Z 62.125,A 180.000,B 0.000,C 180.000} C_DIS
LIN {X 85.901,Y 87.994,Z 62.123,A 180.000,B 0.000,C 180.000} C_DIS
LIN {X 85.850,Y 88.054,Z 62.120,A 180.000,B 0.000,C 180.000} C_DIS
LIN {X 85.799,Y 88.114,Z 62.117,A 180.000,B 0.000,C 180.000} C_DIS
LIN {X 85.750,Y 88.176,Z 62.114,A 180.000,B 0.000,C 180.000} C_DIS
LIN {X 85.703,Y 88.239,Z 62.112,A 180.000,B 0.000,C 180.000} C_DIS
LIN {X 85.655,Y 88.302,Z 62.109,A 180.000,B 0.000,C 180.000} C_DIS
LIN {X 85.608,Y 88.365,Z 62.106,A 180.000,B 0.000,C 180.000} C_DIS
LIN {X 85.561,Y 88.428,Z 62.103,A 180.000,B 0.000,C 180.000} C_DIS
LIN {X 85.513,Y 88.490,Z 62.101,A 180.000,B 0.000,C 180.000} C_DIS
LIN {X 85.466,Y 88.553,Z 62.098,A 180.000,B 0.000,C 180.000} C_DIS
LIN {X 85.419,Y 88.616,Z 62.095,A 180.000,B 0.000,C 180.000} C_DIS
LIN {X 85.371,Y 88.679,Z 62.092,A 180.000,B 0.000,C 180.000} C_DIS
LIN {X 85.324,Y 88.742,Z 62.090,A 180.000,B 0.000,C 180.000} C_DIS
LIN {X 85.277,Y 88.805,Z 62.087,A 180.000,B 0.000,C 180.000} C_DIS
LIN {X 85.232,Y 88.870,Z 62.084,A 180.000,B 0.000,C 180.000} C_DIS
LIN {X 85.188,Y 88.935,Z 62.082,A 180.000,B 0.000,C 180.000} C_DIS
LIN {X 85.144,Y 89.001,Z 62.079,A 180.000,B 0.000,C 180.000} C_DIS
LIN {X 85.101,Y 89.066,Z 62.077,A 180.000,B 0.000,C 180.000} C_DIS
LIN {X 85.057,Y 89.132,Z 62.074,A 180.000,B 0.000,C 180.000} C_DIS
LIN {X 84.969,Y 89.263,Z 62.069,A 180.000,B 0.000,C 180.000} C_DIS
LIN {X 84.882,Y 89.394,Z 62.064,A 180.000,B 0.000,C 180.000} C_DIS
LIN {X 84.795,Y 89.525,Z 62.060,A 180.000,B 0.000,C 180.000} C_DIS
LIN {X 84.715,Y 89.661,Z 62.055,A 180.000,B 0.000,C 180.000} C_DIS
LIN {X 84.635,Y 89.796,Z 62.051,A 180.000,B 0.000,C 180.000} C_DIS
LIN {X 84.555,Y 89.932,Z 62.047,A 180.000,B 0.000,C 180.000} C_DIS
LIN {X 84.475,Y 90.068,Z 62.042,A 180.000,B 0.000,C 180.000} C_DIS
LIN {X 84.395,Y 90.203,Z 62.039,A 180.000,B 0.000,C 180.000} C_DIS
LIN {X 84.320,Y 90.342,Z 62.035,A 180.000,B 0.000,C 180.000} C_DIS
LIN {X 84.248,Y 90.482,Z 62.031,A 180.000,B 0.000,C 180.000} C_DIS
LIN {X 84.175,Y 90.622,Z 62.028,A 180.000,B 0.000,C 180.000} C_DIS
LIN {X 84.103,Y 90.762,Z 62.024,A 180.000,B 0.000,C 180.000} C_DIS
LIN {X 84.031,Y 90.902,Z 62.021,A 180.000,B 0.000,C 180.000} C_DIS
LIN {X 83.961,Y 91.043,Z 62.019,A 180.000,B 0.000,C 180.000} C_DIS
LIN {X 83.897,Y 91.187,Z 62.016,A 180.000,B 0.000,C 180.000} C_DIS
LIN {X 83.768,Y 91.474,Z 62.011,A 180.000,B 0.000,C 180.000} C_DIS
LIN {X 83.641,Y 91.762,Z 62.007,A 180.000,B 0.000,C 180.000} C_DIS
LIN {X 83.528,Y 92.056,Z 62.004,A 180.000,B 0.000,C 180.000} C_DIS
LIN {X 83.415,Y 92.351,Z 62.002,A 180.000,B 0.000,C 180.000} C_DIS
LIN {X 83.308,Y 92.647,Z 62.000,A 180.000,B 0.000,C 180.000} C_DIS
LIN {X 83.226,Y 92.905,Z 62.000,A 180.000,B 0.000,C 180.000} C_DIS
; Cutting Move Starts
LIN {X 83.131,Y 93.203,Z 62.000,A 180.000,B 0.000,C 180.000} C_DIS
LIN {X 83.094,Y 93.321,Z 62.000,A 180.000,B 0.000,C 180.000} C_DIS
LIN {X 83.046,Y 93.500,Z 62.000,A 180.000,B 0.000,C 180.000} C_DIS
LIN {X 82.908,Y 94.036,Z 62.000,A 180.000,B 0.000,C 180.000} C_DIS
LIN {X 82.865,Y 94.215,Z 62.000,A 180.000,B 0.000,C 180.000} C_DIS
LIN {X 82.829,Y 94.394,Z 62.000,A 180.000,B 0.000,C 180.000} C_DIS
LIN {X 82.758,Y 94.751,Z 62.000,A 180.000,B 0.000,C 180.000} C_DIS
LIN {X 82.722,Y 94.930,Z 62.000,A 180.000,B 0.000,C 180.000} C_DIS
LIN {X 82.694,Y 95.109,Z 62.000,A 180.000,B 0.000,C 180.000} C_DIS
LIN {X 82.618,Y 95.645,Z 62.000,A 180.000,B 0.000,C 180.000} C_DIS
LIN {X 82.595,Y 95.815,Z 62.000,A 180.000,B 0.000,C 180.000} C_DIS
LIN {X 82.594,Y 95.824,Z 62.000,A 180.000,B 0.000,C 180.000} C_DIS
LIN {X 82.578,Y 96.003,Z 62.000,A 180.000,B 0.000,C 180.000} C_DIS
LIN {X 82.533,Y 96.539,Z 62.000,A 180.000,B 0.000,C 180.000} C_DIS
LIN {X 82.521,Y 96.718,Z 62.000,A 180.000,B 0.000,C 180.000} C_DIS
LIN {X 82.516,Y 96.897,Z 62.000,A 180.000,B 0.000,C 180.000} C_DIS
LIN {X 82.501,Y 97.433,Z 62.000,A 180.000,B 0.000,C 180.000} C_DIS
LIN {X 82.502,Y 97.612,Z 62.000,A 180.000,B 0.000,C 180.000} C_DIS
LIN {X 82.517,Y 98.148,Z 62.000,A 180.000,B 0.000,C 180.000} C_DIS
LIN {X 82.523,Y 98.327,Z 62.000,A 180.000,B 0.000,C 180.000} C_DIS
LIN {X 82.536,Y 98.505,Z 62.000,A 180.000,B 0.000,C 180.000} C_DIS
LIN {X 82.582,Y 99.042,Z 62.000,A 180.000,B 0.000,C 180.000} C_DIS
LIN {X 82.595,Y 99.185,Z 62.000,A 180.000,B 0.000,C 180.000} C_DIS
LIN {X 82.599,Y 99.221,Z 62.000,A 180.000,B 0.000,C 180.000} C_DIS
LIN {X 82.624,Y 99.399,Z 62.000,A 180.000,B 0.000,C 180.000} C_DIS
LIN {X 82.700,Y 99.936,Z 62.000,A 180.000,B 0.000,C 180.000} C_DIS
LIN {X 82.731,Y 100.114,Z 62.000,A 180.000,B 0.000,C 180.000} C_DIS
LIN {X 82.838,Y 100.651,Z 62.000,A 180.000,B 0.000,C 180.000} C_DIS
LIN {X 82.874,Y 100.829,Z 62.000,A 180.000,B 0.000,C 180.000} C_DIS
LIN {X 82.919,Y 101.008,Z 62.000,A 180.000,B 0.000,C 180.000} C_DIS
LIN {X 83.057,Y 101.545,Z 62.000,A 180.000,B 0.000,C 180.000} C_DIS
LIN {X 83.108,Y 101.723,Z 62.000,A 180.000,B 0.000,C 180.000} C_DIS
LIN {X 83.310,Y 102.358,Z 62.000,A 180.000,B 0.000,C 180.000} C_DIS
LIN {X 83.336,Y 102.438,Z 62.000,A 180.000,B 0.000,C 180.000} C_DIS
LIN {X 83.403,Y 102.617,Z 62.000,A 180.000,B 0.000,C 180.000} C_DIS
LIN {X 83.608,Y 103.153,Z 62.000,A 180.000,B 0.000,C 180.000} C_DIS
LIN {X 83.668,Y 103.300,Z 62.000,A 180.000,B 0.000,C 180.000} C_DIS
LIN {X 83.922,Y 103.869,Z 62.000,A 180.000,B 0.000,C 180.000} C_DIS
LIN {X 84.005,Y 104.047,Z 62.000,A 180.000,B 0.000,C 180.000} C_DIS
LIN {X 84.025,Y 104.087,Z 62.000,A 180.000,B 0.000,C 180.000} C_DIS
LIN {X 84.282,Y 104.584,Z 62.000,A 180.000,B 0.000,C 180.000} C_DIS
LIN {X 84.375,Y 104.762,Z 62.000,A 180.000,B 0.000,C 180.000} C_DIS
LIN {X 84.383,Y 104.775,Z 62.000,A 180.000,B 0.000,C 180.000} C_DIS
LIN {X 84.480,Y 104.941,Z 62.000,A 180.000,B 0.000,C 180.000} C_DIS
LIN {X 84.740,Y 105.382,Z 62.000,A 180.000,B 0.000,C 180.000} C_DIS
LIN {X 84.797,Y 105.477,Z 62.000,A 180.000,B 0.000,C 180.000} C_DIS
LIN {X 84.915,Y 105.656,Z 62.000,A 180.000,B 0.000,C 180.000} C_DIS
LIN {X 85.154,Y 106.014,Z 62.000,A 180.000,B 0.000,C 180.000} C_DIS
LIN {X 85.276,Y 106.193,Z 62.000,A 180.000,B 0.000,C 180.000} C_DIS
LIN {X 85.276,Y 106.194,Z 62.000,A 180.000,B 0.000,C 180.000} C_DIS
LIN {X 85.409,Y 106.371,Z 62.000,A 180.000,B 0.000,C 180.000} C_DIS
LIN {X 85.678,Y 106.729,Z 62.000,A 180.000,B 0.000,C 180.000} C_DIS
LIN {X 85.813,Y 106.902,Z 62.000,A 180.000,B 0.000,C 180.000} C_DIS
LIN {X 85.818,Y 106.908,Z 62.000,A 180.000,B 0.000,C 180.000} C_DIS
LIN {X 86.271,Y 107.444,Z 62.000,A 180.000,B 0.000,C 180.000} C_DIS
LIN {X 86.349,Y 107.532,Z 62.000,A 180.000,B 0.000,C 180.000} C_DIS
LIN {X 86.435,Y 107.623,Z 62.000,A 180.000,B 0.000,C 180.000} C_DIS
LIN {X 86.773,Y 107.980,Z 62.000,A 180.000,B 0.000,C 180.000} C_DIS
LIN {X 86.885,Y 108.099,Z 62.000,A 180.000,B 0.000,C 180.000} C_DIS
LIN {X 86.947,Y 108.159,Z 62.000,A 180.000,B 0.000,C 180.000} C_DIS
LIN {X 87.422,Y 108.607,Z 62.000,A 180.000,B 0.000,C 180.000} C_DIS
LIN {X 87.517,Y 108.695,Z 62.000,A 180.000,B 0.000,C 180.000} C_DIS
LIN {X 87.601,Y 108.767,Z 62.000,A 180.000,B 0.000,C 180.000} C_DIS
LIN {X 87.958,Y 109.069,Z 62.000,A 180.000,B 0.000,C 180.000} C_DIS
LIN {X 88.137,Y 109.219,Z 62.000,A 180.000,B 0.000,C 180.000} C_DIS
LIN {X 88.153,Y 109.232,Z 62.000,A 180.000,B 0.000,C 180.000} C_DIS
LIN {X 88.316,Y 109.355,Z 62.000,A 180.000,B 0.000,C 180.000} C_DIS
LIN {X 88.673,Y 109.624,Z 62.000,A 180.000,B 0.000,C 180.000} C_DIS
LIN {X 88.852,Y 109.756,Z 62.000,A 180.000,B 0.000,C 180.000} C_DIS
LIN {X 88.870,Y 109.768,Z 62.000,A 180.000,B 0.000,C 180.000} C_DIS
LIN {X 89.031,Y 109.875,Z 62.000,A 180.000,B 0.000,C 180.000} C_DIS
LIN {X 89.405,Y 110.126,Z 62.000,A 180.000,B 0.000,C 180.000} C_DIS
LIN {X 89.567,Y 110.230,Z 62.000,A 180.000,B 0.000,C 180.000} C_DIS
LIN {X 89.693,Y 110.304,Z 62.000,A 180.000,B 0.000,C 180.000} C_DIS
LIN {X 90.103,Y 110.546,Z 62.000,A 180.000,B 0.000,C 180.000} C_DIS
LIN {X 90.282,Y 110.649,Z 62.000,A 180.000,B 0.000,C 180.000} C_DIS
LIN {X 90.307,Y 110.662,Z 62.000,A 180.000,B 0.000,C 180.000} C_DIS
LIN {X 90.818,Y 110.926,Z 62.000,A 180.000,B 0.000,C 180.000} C_DIS
LIN {X 90.997,Y 111.017,Z 62.000,A 180.000,B 0.000,C 180.000} C_DIS
LIN {X 91.002,Y 111.019,Z 62.000,A 180.000,B 0.000,C 180.000} C_DIS
LIN {X 91.176,Y 111.098,Z 62.000,A 180.000,B 0.000,C 180.000} C_DIS
LIN {X 91.533,Y 111.258,Z 62.000,A 180.000,B 0.000,C 180.000} C_DIS
LIN {X 91.712,Y 111.338,Z 62.000,A 180.000,B 0.000,C 180.000} C_DIS
LIN {X 91.806,Y 111.377,Z 62.000,A 180.000,B 0.000,C 180.000} C_DIS
LIN {X 91.891,Y 111.409,Z 62.000,A 180.000,B 0.000,C 180.000} C_DIS
LIN {X 92.427,Y 111.614,Z 62.000,A 180.000,B 0.000,C 180.000} C_DIS
LIN {X 92.606,Y 111.678,Z 62.000,A 180.000,B 0.000,C 180.000} C_DIS
LIN {X 92.964,Y 111.792,Z 62.000,A 180.000,B 0.000,C 180.000} C_DIS
LIN {X 93.142,Y 111.849,Z 62.000,A 180.000,B 0.000,C 180.000} C_DIS
LIN {X 93.321,Y 111.906,Z 62.000,A 180.000,B 0.000,C 180.000} C_DIS
LIN {X 93.346,Y 111.913,Z 62.000,A 180.000,B 0.000,C 180.000} C_DIS
LIN {X 93.500,Y 111.954,Z 62.000,A 180.000,B 0.000,C 180.000} C_DIS
LIN {X 94.036,Y 112.092,Z 62.000,A 180.000,B 0.000,C 180.000} C_DIS
LIN {X 94.215,Y 112.135,Z 62.000,A 180.000,B 0.000,C 180.000} C_DIS
LIN {X 94.394,Y 112.171,Z 62.000,A 180.000,B 0.000,C 180.000} C_DIS
LIN {X 94.895,Y 112.271,Z 62.000,A 180.000,B 0.000,C 180.000} C_DIS
LIN {X 94.930,Y 112.278,Z 62.000,A 180.000,B 0.000,C 180.000} C_DIS
LIN {X 95.109,Y 112.306,Z 62.000,A 180.000,B 0.000,C 180.000} C_DIS
LIN {X 95.645,Y 112.382,Z 62.000,A 180.000,B 0.000,C 180.000} C_DIS
LIN {X 95.824,Y 112.406,Z 62.000,A 180.000,B 0.000,C 180.000} C_DIS
LIN {X 96.003,Y 112.422,Z 62.000,A 180.000,B 0.000,C 180.000} C_DIS
LIN {X 96.539,Y 112.467,Z 62.000,A 180.000,B 0.000,C 180.000} C_DIS
LIN {X 96.718,Y 112.479,Z 62.000,A 180.000,B 0.000,C 180.000} C_DIS
LIN {X 96.897,Y 112.484,Z 62.000,A 180.000,B 0.000,C 180.000} C_DIS
LIN {X 97.433,Y 112.499,Z 62.000,A 180.000,B 0.000,C 180.000} C_DIS
LIN {X 97.612,Y 112.498,Z 62.000,A 180.000,B 0.000,C 180.000} C_DIS
LIN {X 98.148,Y 112.483,Z 62.000,A 180.000,B 0.000,C 180.000} C_DIS
LIN {X 98.327,Y 112.477,Z 62.000,A 180.000,B 0.000,C 180.000} C_DIS
LIN {X 98.505,Y 112.464,Z 62.000,A 180.000,B 0.000,C 180.000} C_DIS
LIN {X 99.042,Y 112.418,Z 62.000,A 180.000,B 0.000,C 180.000} C_DIS
LIN {X 99.221,Y 112.401,Z 62.000,A 180.000,B 0.000,C 180.000} C_DIS
LIN {X 99.399,Y 112.376,Z 62.000,A 180.000,B 0.000,C 180.000} C_DIS
LIN {X 99.936,Y 112.300,Z 62.000,A 180.000,B 0.000,C 180.000} C_DIS
LIN {X 100.105,Y 112.271,Z 62.000,A 180.000,B 0.000,C 180.000} C_DIS
LIN {X 100.651,Y 112.162,Z 62.000,A 180.000,B 0.000,C 180.000} C_DIS
LIN {X 100.829,Y 112.126,Z 62.000,A 180.000,B 0.000,C 180.000} C_DIS
LIN {X 100.966,Y 112.092,Z 62.000,A 180.000,B 0.000,C 180.000} C_DIS
LIN {X 101.545,Y 111.943,Z 62.000,A 180.000,B 0.000,C 180.000} C_DIS
LIN {X 101.654,Y 111.913,Z 62.000,A 180.000,B 0.000,C 180.000} C_DIS
LIN {X 101.723,Y 111.892,Z 62.000,A 180.000,B 0.000,C 180.000} C_DIS
LIN {X 102.260,Y 111.721,Z 62.000,A 180.000,B 0.000,C 180.000} C_DIS
LIN {X 102.438,Y 111.664,Z 62.000,A 180.000,B 0.000,C 180.000} C_DIS
LIN {X 102.617,Y 111.597,Z 62.000,A 180.000,B 0.000,C 180.000} C_DIS
LIN {X 103.153,Y 111.392,Z 62.000,A 180.000,B 0.000,C 180.000} C_DIS
LIN {X 103.194,Y 111.377,Z 62.000,A 180.000,B 0.000,C 180.000} C_DIS
LIN {X 103.332,Y 111.318,Z 62.000,A 180.000,B 0.000,C 180.000} C_DIS
LIN {X 103.869,Y 111.078,Z 62.000,A 180.000,B 0.000,C 180.000} C_DIS
LIN {X 103.998,Y 111.019,Z 62.000,A 180.000,B 0.000,C 180.000} C_DIS
LIN {X 104.047,Y 110.995,Z 62.000,A 180.000,B 0.000,C 180.000} C_DIS
LIN {X 104.226,Y 110.903,Z 62.000,A 180.000,B 0.000,C 180.000} C_DIS
LIN {X 104.693,Y 110.662,Z 62.000,A 180.000,B 0.000,C 180.000} C_DIS
LIN {X 104.762,Y 110.625,Z 62.000,A 180.000,B 0.000,C 180.000} C_DIS
LIN {X 104.941,Y 110.520,Z 62.000,A 180.000,B 0.000,C 180.000} C_DIS
LIN {X 105.307,Y 110.304,Z 62.000,A 180.000,B 0.000,C 180.000} C_DIS
LIN {X 105.477,Y 110.203,Z 62.000,A 180.000,B 0.000,C 180.000} C_DIS
LIN {X 105.595,Y 110.126,Z 62.000,A 180.000,B 0.000,C 180.000} C_DIS
LIN {X 106.014,Y 109.846,Z 62.000,A 180.000,B 0.000,C 180.000} C_DIS
LIN {X 106.130,Y 109.768,Z 62.000,A 180.000,B 0.000,C 180.000} C_DIS
LIN {X 106.193,Y 109.724,Z 62.000,A 180.000,B 0.000,C 180.000} C_DIS
LIN {X 106.371,Y 109.591,Z 62.000,A 180.000,B 0.000,C 180.000} C_DIS
LIN {X 106.729,Y 109.322,Z 62.000,A 180.000,B 0.000,C 180.000} C_DIS
LIN {X 106.847,Y 109.232,Z 62.000,A 180.000,B 0.000,C 180.000} C_DIS
LIN {X 106.908,Y 109.182,Z 62.000,A 180.000,B 0.000,C 180.000} C_DIS
LIN {X 107.444,Y 108.729,Z 62.000,A 180.000,B 0.000,C 180.000} C_DIS
LIN {X 107.483,Y 108.695,Z 62.000,A 180.000,B 0.000,C 180.000} C_DIS
LIN {X 107.623,Y 108.565,Z 62.000,A 180.000,B 0.000,C 180.000} C_DIS
LIN {X 108.053,Y 108.159,Z 62.000,A 180.000,B 0.000,C 180.000} C_DIS
LIN {X 108.159,Y 108.053,Z 62.000,A 180.000,B 0.000,C 180.000} C_DIS
LIN {X 108.565,Y 107.623,Z 62.000,A 180.000,B 0.000,C 180.000} C_DIS
LIN {X 108.695,Y 107.483,Z 62.000,A 180.000,B 0.000,C 180.000} C_DIS
LIN {X 108.729,Y 107.444,Z 62.000,A 180.000,B 0.000,C 180.000} C_DIS
LIN {X 109.182,Y 106.908,Z 62.000,A 180.000,B 0.000,C 180.000} C_DIS
LIN {X 109.232,Y 106.847,Z 62.000,A 180.000,B 0.000,C 180.000} C_DIS
LIN {X 109.322,Y 106.729,Z 62.000,A 180.000,B 0.000,C 180.000} C_DIS
LIN {X 109.591,Y 106.371,Z 62.000,A 180.000,B 0.000,C 180.000} C_DIS
LIN {X 109.724,Y 106.193,Z 62.000,A 180.000,B 0.000,C 180.000} C_DIS
LIN {X 109.768,Y 106.130,Z 62.000,A 180.000,B 0.000,C 180.000} C_DIS
LIN {X 109.846,Y 106.014,Z 62.000,A 180.000,B 0.000,C 180.000} C_DIS
LIN {X 110.126,Y 105.595,Z 62.000,A 180.000,B 0.000,C 180.000} C_DIS
LIN {X 110.203,Y 105.477,Z 62.000,A 180.000,B 0.000,C 180.000} C_DIS
LIN {X 110.304,Y 105.307,Z 62.000,A 180.000,B 0.000,C 180.000} C_DIS
LIN {X 110.520,Y 104.941,Z 62.000,A 180.000,B 0.000,C 180.000} C_DIS
LIN {X 110.625,Y 104.762,Z 62.000,A 180.000,B 0.000,C 180.000} C_DIS
LIN {X 110.662,Y 104.693,Z 62.000,A 180.000,B 0.000,C 180.000} C_DIS
LIN {X 110.903,Y 104.226,Z 62.000,A 180.000,B 0.000,C 180.000} C_DIS
LIN {X 110.995,Y 104.047,Z 62.000,A 180.000,B 0.000,C 180.000} C_DIS
LIN {X 111.019,Y 103.998,Z 62.000,A 180.000,B 0.000,C 180.000} C_DIS
LIN {X 111.078,Y 103.869,Z 62.000,A 180.000,B 0.000,C 180.000} C_DIS
LIN {X 111.318,Y 103.332,Z 62.000,A 180.000,B 0.000,C 180.000} C_DIS
LIN {X 111.377,Y 103.194,Z 62.000,A 180.000,B 0.000,C 180.000} C_DIS
LIN {X 111.392,Y 103.153,Z 62.000,A 180.000,B 0.000,C 180.000} C_DIS
LIN {X 111.597,Y 102.617,Z 62.000,A 180.000,B 0.000,C 180.000} C_DIS
LIN {X 111.664,Y 102.438,Z 62.000,A 180.000,B 0.000,C 180.000} C_DIS
LIN {X 111.721,Y 102.260,Z 62.000,A 180.000,B 0.000,C 180.000} C_DIS
LIN {X 111.892,Y 101.723,Z 62.000,A 180.000,B 0.000,C 180.000} C_DIS
LIN {X 111.913,Y 101.654,Z 62.000,A 180.000,B 0.000,C 180.000} C_DIS
LIN {X 111.943,Y 101.545,Z 62.000,A 180.000,B 0.000,C 180.000} C_DIS
LIN {X 112.092,Y 100.966,Z 62.000,A 180.000,B 0.000,C 180.000} C_DIS
LIN {X 112.126,Y 100.829,Z 62.000,A 180.000,B 0.000,C 180.000} C_DIS
LIN {X 112.162,Y 100.651,Z 62.000,A 180.000,B 0.000,C 180.000} C_DIS
LIN {X 112.271,Y 100.105,Z 62.000,A 180.000,B 0.000,C 180.000} C_DIS
LIN {X 112.300,Y 99.936,Z 62.000,A 180.000,B 0.000,C 180.000} C_DIS
LIN {X 112.376,Y 99.399,Z 62.000,A 180.000,B 0.000,C 180.000} C_DIS
LIN {X 112.401,Y 99.221,Z 62.000,A 180.000,B 0.000,C 180.000} C_DIS
LIN {X 112.418,Y 99.042,Z 62.000,A 180.000,B 0.000,C 180.000} C_DIS
LIN {X 112.464,Y 98.505,Z 62.000,A 180.000,B 0.000,C 180.000} C_DIS
LIN {X 112.477,Y 98.327,Z 62.000,A 180.000,B 0.000,C 180.000} C_DIS
LIN {X 112.483,Y 98.148,Z 62.000,A 180.000,B 0.000,C 180.000} C_DIS
LIN {X 112.498,Y 97.612,Z 62.000,A 180.000,B 0.000,C 180.000} C_DIS
LIN {X 112.499,Y 97.433,Z 62.000,A 180.000,B 0.000,C 180.000} C_DIS
LIN {X 112.484,Y 96.897,Z 62.000,A 180.000,B 0.000,C 180.000} C_DIS
LIN {X 112.479,Y 96.718,Z 62.000,A 180.000,B 0.000,C 180.000} C_DIS
LIN {X 112.467,Y 96.539,Z 62.000,A 180.000,B 0.000,C 180.000} C_DIS
LIN {X 112.422,Y 96.003,Z 62.000,A 180.000,B 0.000,C 180.000} C_DIS
LIN {X 112.406,Y 95.824,Z 62.000,A 180.000,B 0.000,C 180.000} C_DIS
LIN {X 112.382,Y 95.645,Z 62.000,A 180.000,B 0.000,C 180.000} C_DIS
LIN {X 112.306,Y 95.109,Z 62.000,A 180.000,B 0.000,C 180.000} C_DIS
LIN {X 112.278,Y 94.930,Z 62.000,A 180.000,B 0.000,C 180.000} C_DIS
LIN {X 112.271,Y 94.895,Z 62.000,A 180.000,B 0.000,C 180.000} C_DIS
LIN {X 112.171,Y 94.394,Z 62.000,A 180.000,B 0.000,C 180.000} C_DIS
LIN {X 112.135,Y 94.215,Z 62.000,A 180.000,B 0.000,C 180.000} C_DIS
LIN {X 112.092,Y 94.036,Z 62.000,A 180.000,B 0.000,C 180.000} C_DIS
LIN {X 111.954,Y 93.500,Z 62.000,A 180.000,B 0.000,C 180.000} C_DIS
LIN {X 111.913,Y 93.346,Z 62.000,A 180.000,B 0.000,C 180.000} C_DIS
LIN {X 111.906,Y 93.321,Z 62.000,A 180.000,B 0.000,C 180.000} C_DIS
LIN {X 111.849,Y 93.142,Z 62.000,A 180.000,B 0.000,C 180.000} C_DIS
LIN {X 111.734,Y 92.782,Z 62.000,A 180.000,B 0.000,C 180.000} C_DIS
LIN {X 111.678,Y 92.606,Z 62.000,A 180.000,B 0.000,C 180.000} C_DIS
LIN {X 111.614,Y 92.427,Z 62.000,A 180.000,B 0.000,C 180.000} C_DIS
LIN {X 111.409,Y 91.891,Z 62.000,A 180.000,B 0.000,C 180.000} C_DIS
LIN {X 111.377,Y 91.806,Z 62.000,A 180.000,B 0.000,C 180.000} C_DIS
LIN {X 111.338,Y 91.712,Z 62.000,A 180.000,B 0.000,C 180.000} C_DIS
LIN {X 111.258,Y 91.533,Z 62.000,A 180.000,B 0.000,C 180.000} C_DIS
LIN {X 111.098,Y 91.176,Z 62.000,A 180.000,B 0.000,C 180.000} C_DIS
LIN {X 111.019,Y 91.002,Z 62.000,A 180.000,B 0.000,C 180.000} C_DIS
LIN {X 111.017,Y 90.997,Z 62.000,A 180.000,B 0.000,C 180.000} C_DIS
LIN {X 110.926,Y 90.818,Z 62.000,A 180.000,B 0.000,C 180.000} C_DIS
LIN {X 110.662,Y 90.307,Z 62.000,A 180.000,B 0.000,C 180.000} C_DIS
LIN {X 110.649,Y 90.282,Z 62.000,A 180.000,B 0.000,C 180.000} C_DIS
LIN {X 110.546,Y 90.103,Z 62.000,A 180.000,B 0.000,C 180.000} C_DIS
LIN {X 110.304,Y 89.693,Z 62.000,A 180.000,B 0.000,C 180.000} C_DIS
LIN {X 110.230,Y 89.567,Z 62.000,A 180.000,B 0.000,C 180.000} C_DIS
LIN {X 110.126,Y 89.405,Z 62.000,A 180.000,B 0.000,C 180.000} C_DIS
LIN {X 109.875,Y 89.031,Z 62.000,A 180.000,B 0.000,C 180.000} C_DIS
LIN {X 109.768,Y 88.870,Z 62.000,A 180.000,B 0.000,C 180.000} C_DIS
LIN {X 109.756,Y 88.852,Z 62.000,A 180.000,B 0.000,C 180.000} C_DIS
LIN {X 109.624,Y 88.673,Z 62.000,A 180.000,B 0.000,C 180.000} C_DIS
LIN {X 109.355,Y 88.316,Z 62.000,A 180.000,B 0.000,C 180.000} C_DIS
LIN {X 109.232,Y 88.153,Z 62.000,A 180.000,B 0.000,C 180.000} C_DIS
LIN {X 109.219,Y 88.137,Z 62.000,A 180.000,B 0.000,C 180.000} C_DIS
LIN {X 109.069,Y 87.958,Z 62.000,A 180.000,B 0.000,C 180.000} C_DIS
LIN {X 108.767,Y 87.601,Z 62.000,A 180.000,B 0.000,C 180.000} C_DIS
LIN {X 108.695,Y 87.517,Z 62.000,A 180.000,B 0.000,C 180.000} C_DIS
LIN {X 108.607,Y 87.422,Z 62.000,A 180.000,B 0.000,C 180.000} C_DIS
LIN {X 108.159,Y 86.947,Z 62.000,A 180.000,B 0.000,C 180.000} C_DIS
LIN {X 108.099,Y 86.885,Z 62.000,A 180.000,B 0.000,C 180.000} C_DIS
LIN {X 107.980,Y 86.773,Z 62.000,A 180.000,B 0.000,C 180.000} C_DIS
LIN {X 107.623,Y 86.435,Z 62.000,A 180.000,B 0.000,C 180.000} C_DIS
LIN {X 107.532,Y 86.349,Z 62.000,A 180.000,B 0.000,C 180.000} C_DIS
LIN {X 107.444,Y 86.271,Z 62.000,A 180.000,B 0.000,C 180.000} C_DIS
LIN {X 106.908,Y 85.818,Z 62.000,A 180.000,B 0.000,C 180.000} C_DIS
LIN {X 106.902,Y 85.813,Z 62.000,A 180.000,B 0.000,C 180.000} C_DIS
LIN {X 106.729,Y 85.678,Z 62.000,A 180.000,B 0.000,C 180.000} C_DIS
LIN {X 106.371,Y 85.409,Z 62.000,A 180.000,B 0.000,C 180.000} C_DIS
LIN {X 106.194,Y 85.276,Z 62.000,A 180.000,B 0.000,C 180.000} C_DIS
LIN {X 106.193,Y 85.276,Z 62.000,A 180.000,B 0.000,C 180.000} C_DIS
LIN {X 106.014,Y 85.154,Z 62.000,A 180.000,B 0.000,C 180.000} C_DIS
LIN {X 105.656,Y 84.915,Z 62.000,A 180.000,B 0.000,C 180.000} C_DIS
LIN {X 105.477,Y 84.797,Z 62.000,A 180.000,B 0.000,C 180.000} C_DIS
LIN {X 105.382,Y 84.740,Z 62.000,A 180.000,B 0.000,C 180.000} C_DIS
LIN {X 104.941,Y 84.480,Z 62.000,A 180.000,B 0.000,C 180.000} C_DIS
LIN {X 104.775,Y 84.383,Z 62.000,A 180.000,B 0.000,C 180.000} C_DIS
LIN {X 104.762,Y 84.375,Z 62.000,A 180.000,B 0.000,C 180.000} C_DIS
LIN {X 104.584,Y 84.282,Z 62.000,A 180.000,B 0.000,C 180.000} C_DIS
LIN {X 104.087,Y 84.025,Z 62.000,A 180.000,B 0.000,C 180.000} C_DIS
LIN {X 104.047,Y 84.005,Z 62.000,A 180.000,B 0.000,C 180.000} C_DIS
LIN {X 103.869,Y 83.922,Z 62.000,A 180.000,B 0.000,C 180.000} C_DIS
LIN {X 103.300,Y 83.668,Z 62.000,A 180.000,B 0.000,C 180.000} C_DIS
LIN {X 103.153,Y 83.608,Z 62.000,A 180.000,B 0.000,C 180.000} C_DIS
LIN {X 102.617,Y 83.403,Z 62.000,A 180.000,B 0.000,C 180.000} C_DIS
LIN {X 102.438,Y 83.336,Z 62.000,A 180.000,B 0.000,C 180.000} C_DIS
LIN {X 102.358,Y 83.310,Z 62.000,A 180.000,B 0.000,C 180.000} C_DIS
LIN {X 101.723,Y 83.108,Z 62.000,A 180.000,B 0.000,C 180.000} C_DIS
LIN {X 101.545,Y 83.057,Z 62.000,A 180.000,B 0.000,C 180.000} C_DIS
LIN {X 101.008,Y 82.919,Z 62.000,A 180.000,B 0.000,C 180.000} C_DIS
LIN {X 100.829,Y 82.874,Z 62.000,A 180.000,B 0.000,C 180.000} C_DIS
LIN {X 100.651,Y 82.838,Z 62.000,A 180.000,B 0.000,C 180.000} C_DIS
LIN {X 100.114,Y 82.731,Z 62.000,A 180.000,B 0.000,C 180.000} C_DIS
LIN {X 99.936,Y 82.700,Z 62.000,A 180.000,B 0.000,C 180.000} C_DIS
LIN {X 99.399,Y 82.624,Z 62.000,A 180.000,B 0.000,C 180.000} C_DIS
LIN {X 99.221,Y 82.599,Z 62.000,A 180.000,B 0.000,C 180.000} C_DIS
LIN {X 99.185,Y 82.595,Z 62.000,A 180.000,B 0.000,C 180.000} C_DIS
LIN {X 99.042,Y 82.582,Z 62.000,A 180.000,B 0.000,C 180.000} C_DIS
LIN {X 98.505,Y 82.536,Z 62.000,A 180.000,B 0.000,C 180.000} C_DIS
LIN {X 98.327,Y 82.523,Z 62.000,A 180.000,B 0.000,C 180.000} C_DIS
LIN {X 98.148,Y 82.517,Z 62.000,A 180.000,B 0.000,C 180.000} C_DIS
LIN {X 97.612,Y 82.502,Z 62.000,A 180.000,B 0.000,C 180.000} C_DIS
LIN {X 97.433,Y 82.501,Z 62.000,A 180.000,B 0.000,C 180.000} C_DIS
LIN {X 97.153,Y 82.509,Z 62.000,A 180.000,B 0.000,C 180.000} C_DIS
LIN {X 96.897,Y 82.516,Z 62.000,A 180.000,B 0.000,C 180.000} C_DIS
LIN {X 96.718,Y 82.521,Z 62.000,A 180.000,B 0.000,C 180.000} C_DIS
LIN {X 96.539,Y 82.533,Z 62.000,A 180.000,B 0.000,C 180.000} C_DIS
LIN {X 96.003,Y 82.578,Z 62.000,A 180.000,B 0.000,C 180.000} C_DIS
LIN {X 95.824,Y 82.594,Z 62.000,A 180.000,B 0.000,C 180.000} C_DIS
LIN {X 95.815,Y 82.595,Z 62.000,A 180.000,B 0.000,C 180.000} C_DIS
LIN {X 95.645,Y 82.618,Z 62.000,A 180.000,B 0.000,C 180.000} C_DIS
LIN {X 95.109,Y 82.694,Z 62.000,A 180.000,B 0.000,C 180.000} C_DIS
LIN {X 94.930,Y 82.722,Z 62.000,A 180.000,B 0.000,C 180.000} C_DIS
LIN {X 94.751,Y 82.758,Z 62.000,A 180.000,B 0.000,C 180.000} C_DIS
LIN {X 94.394,Y 82.829,Z 62.000,A 180.000,B 0.000,C 180.000} C_DIS
LIN {X 94.215,Y 82.865,Z 62.000,A 180.000,B 0.000,C 180.000} C_DIS
LIN {X 94.036,Y 82.908,Z 62.000,A 180.000,B 0.000,C 180.000} C_DIS
LIN {X 93.500,Y 83.046,Z 62.000,A 180.000,B 0.000,C 180.000} C_DIS
LIN {X 93.321,Y 83.094,Z 62.000,A 180.000,B 0.000,C 180.000} C_DIS
LIN {X 93.203,Y 83.131,Z 62.000,A 180.000,B 0.000,C 180.000} C_DIS
LIN {X 92.642,Y 83.310,Z 62.000,A 180.000,B 0.000,C 180.000} C_DIS
LIN {X 92.606,Y 83.322,Z 62.000,A 180.000,B 0.000,C 180.000} C_DIS
LIN {X 92.427,Y 83.386,Z 62.000,A 180.000,B 0.000,C 180.000} C_DIS
LIN {X 91.891,Y 83.591,Z 62.000,A 180.000,B 0.000,C 180.000} C_DIS
LIN {X 91.712,Y 83.662,Z 62.000,A 180.000,B 0.000,C 180.000} C_DIS
LIN {X 91.700,Y 83.668,Z 62.000,A 180.000,B 0.000,C 180.000} C_DIS
LIN {X 91.176,Y 83.902,Z 62.000,A 180.000,B 0.000,C 180.000} C_DIS
LIN {X 90.997,Y 83.983,Z 62.000,A 180.000,B 0.000,C 180.000} C_DIS
LIN {X 90.913,Y 84.025,Z 62.000,A 180.000,B 0.000,C 180.000} C_DIS
LIN {X 90.461,Y 84.259,Z 62.000,A 180.000,B 0.000,C 180.000} C_DIS
LIN {X 90.282,Y 84.351,Z 62.000,A 180.000,B 0.000,C 180.000} C_DIS
LIN {X 90.225,Y 84.383,Z 62.000,A 180.000,B 0.000,C 180.000} C_DIS
LIN {X 90.103,Y 84.454,Z 62.000,A 180.000,B 0.000,C 180.000} C_DIS
LIN {X 89.618,Y 84.740,Z 62.000,A 180.000,B 0.000,C 180.000} C_DIS
LIN {X 89.567,Y 84.770,Z 62.000,A 180.000,B 0.000,C 180.000} C_DIS
LIN {X 89.388,Y 84.886,Z 62.000,A 180.000,B 0.000,C 180.000} C_DIS
LIN {X 89.031,Y 85.125,Z 62.000,A 180.000,B 0.000,C 180.000} C_DIS
LIN {X 88.852,Y 85.244,Z 62.000,A 180.000,B 0.000,C 180.000} C_DIS
LIN {X 88.806,Y 85.276,Z 62.000,A 180.000,B 0.000,C 180.000} C_DIS
LIN {X 88.673,Y 85.376,Z 62.000,A 180.000,B 0.000,C 180.000} C_DIS
LIN {X 88.316,Y 85.645,Z 62.000,A 180.000,B 0.000,C 180.000} C_DIS
LIN {X 88.137,Y 85.781,Z 62.000,A 180.000,B 0.000,C 180.000} C_DIS
LIN {X 88.098,Y 85.813,Z 62.000,A 180.000,B 0.000,C 180.000} C_DIS
LIN {X 87.779,Y 86.082,Z 62.000,A 180.000,B 0.000,C 180.000} C_DIS
LIN {X 87.601,Y 86.233,Z 62.000,A 180.000,B 0.000,C 180.000} C_DIS
LIN {X 87.468,Y 86.349,Z 62.000,A 180.000,B 0.000,C 180.000} C_DIS
LIN {X 87.422,Y 86.393,Z 62.000,A 180.000,B 0.000,C 180.000} C_DIS
LIN {X 87.064,Y 86.731,Z 62.000,A 180.000,B 0.000,C 180.000} C_DIS
LIN {X 86.901,Y 86.885,Z 62.000,A 180.000,B 0.000,C 180.000} C_DIS
LIN {X 86.885,Y 86.901,Z 62.000,A 180.000,B 0.000,C 180.000} C_DIS
LIN {X 86.731,Y 87.064,Z 62.000,A 180.000,B 0.000,C 180.000} C_DIS
LIN {X 86.393,Y 87.422,Z 62.000,A 180.000,B 0.000,C 180.000} C_DIS
LIN {X 86.349,Y 87.468,Z 62.000,A 180.000,B 0.000,C 180.000} C_DIS
LIN {X 86.233,Y 87.601,Z 62.000,A 180.000,B 0.000,C 180.000} C_DIS
LIN {X 85.931,Y 87.958,Z 62.000,A 180.000,B 0.000,C 180.000} C_DIS
LIN {X 85.813,Y 88.098,Z 62.000,A 180.000,B 0.000,C 180.000} C_DIS
LIN {X 85.781,Y 88.137,Z 62.000,A 180.000,B 0.000,C 180.000} C_DIS
LIN {X 85.645,Y 88.316,Z 62.000,A 180.000,B 0.000,C 180.000} C_DIS
LIN {X 85.376,Y 88.673,Z 62.000,A 180.000,B 0.000,C 180.000} C_DIS
LIN {X 85.276,Y 88.806,Z 62.000,A 180.000,B 0.000,C 180.000} C_DIS
LIN {X 85.244,Y 88.852,Z 62.000,A 180.000,B 0.000,C 180.000} C_DIS
LIN {X 85.125,Y 89.031,Z 62.000,A 180.000,B 0.000,C 180.000} C_DIS
LIN {X 84.886,Y 89.388,Z 62.000,A 180.000,B 0.000,C 180.000} C_DIS
LIN {X 84.770,Y 89.567,Z 62.000,A 180.000,B 0.000,C 180.000} C_DIS
LIN {X 84.740,Y 89.618,Z 62.000,A 180.000,B 0.000,C 180.000} C_DIS
LIN {X 84.454,Y 90.103,Z 62.000,A 180.000,B 0.000,C 180.000} C_DIS
LIN {X 84.383,Y 90.225,Z 62.000,A 180.000,B 0.000,C 180.000} C_DIS
LIN {X 84.351,Y 90.282,Z 62.000,A 180.000,B 0.000,C 180.000} C_DIS
LIN {X 84.259,Y 90.461,Z 62.000,A 180.000,B 0.000,C 180.000} C_DIS
LIN {X 84.025,Y 90.913,Z 62.000,A 180.000,B 0.000,C 180.000} C_DIS
LIN {X 83.983,Y 90.997,Z 62.000,A 180.000,B 0.000,C 180.000} C_DIS
LIN {X 83.902,Y 91.176,Z 62.000,A 180.000,B 0.000,C 180.000} C_DIS
LIN {X 83.668,Y 91.700,Z 62.000,A 180.000,B 0.000,C 180.000} C_DIS
LIN {X 83.662,Y 91.712,Z 62.000,A 180.000,B 0.000,C 180.000} C_DIS
LIN {X 83.591,Y 91.891,Z 62.000,A 180.000,B 0.000,C 180.000} C_DIS
LIN {X 83.386,Y 92.427,Z 62.000,A 180.000,B 0.000,C 180.000} C_DIS
LIN {X 83.322,Y 92.606,Z 62.000,A 180.000,B 0.000,C 180.000} C_DIS
LIN {X 83.310,Y 92.642,Z 62.000,A 180.000,B 0.000,C 180.000} C_DIS
LIN {X 83.226,Y 92.905,Z 62.000,A 180.000,B 0.000,C 180.000} C_DIS
; Lead Out Move Starts
LIN {X 82.901,Y 93.230,Z 62.000,A 180.000,B 0.000,C 180.000} C_DIS
LIN {X 82.448,Y 93.152,Z 62.000,A 180.000,B 0.000,C 180.000} C_DIS
LIN {X 81.718,Y 92.600,Z 62.000,A 180.000,B 0.000,C 180.000} C_DIS
LIN {X 81.437,Y 92.387,Z 62.146,A 180.000,B 0.000,C 180.000} C_DIS
LIN {X 81.320,Y 92.298,Z 62.500,A 180.000,B 0.000,C 180.000} C_DIS
; Rapid Move Starts
LIN {X 81.320,Y 92.298,Z 95.000,A 180.000,B 0.000,C 180.000} C_DIS
LIN {X 67.008,Y 99.176,Z 95.000,A 180.000,B 0.000,C 180.000} C_DIS
LIN {X 67.008,Y 99.176,Z 79.498,A 180.000,B 0.000,C 180.000} C_DIS
; Plunge Move Starts
$VEL.CP=0.01
LIN {X 67.008,Y 99.176,Z 78.625,A 180.000,B 0.000,C 180.000} C_DIS
; Lead In Move Starts
LIN {X 67.008,Y 99.176,Z 77.500,A 180.000,B 0.000,C 180.000} C_DIS
LIN {X 66.870,Y 99.223,Z 77.146,A 180.000,B 0.000,C 180.000} C_DIS
LIN {X 66.535,Y 99.336,Z 77.000,A 180.000,B 0.000,C 180.000} C_DIS
LIN {X 66.246,Y 99.435,Z 77.000,A 180.000,B 0.000,C 180.000} C_DIS
LIN {X 65.864,Y 99.410,Z 77.000,A 180.000,B 0.000,C 180.000} C_DIS
LIN {X 65.612,Y 99.122,Z 77.000,A 180.000,B 0.000,C 180.000} C_DIS
; Cutting Move Starts
$VEL.CP=0.02
LIN {X 65.582,Y 99.042,Z 77.000,A 180.000,B 0.000,C 180.000} C_DIS
LIN {X 65.516,Y 98.863,Z 77.000,A 180.000,B 0.000,C 180.000} C_DIS
LIN {X 65.450,Y 98.684,Z 77.000,A 180.000,B 0.000,C 180.000} C_DIS
LIN {X 65.433,Y 98.640,Z 77.000,A 180.000,B 0.000,C 180.000} C_DIS
LIN {X 65.375,Y 98.505,Z 77.000,A 180.000,B 0.000,C 180.000} C_DIS
LIN {X 65.290,Y 98.327,Z 77.000,A 180.000,B 0.000,C 180.000} C_DIS
LIN {X 65.206,Y 98.148,Z 77.000,A 180.000,B 0.000,C 180.000} C_DIS
LIN {X 65.117,Y 97.969,Z 77.000,A 180.000,B 0.000,C 180.000} C_DIS
LIN {X 65.075,Y 97.896,Z 77.000,A 180.000,B 0.000,C 180.000} C_DIS
LIN {X 64.897,Y 97.592,Z 77.000,A 180.000,B 0.000,C 180.000} C_DIS
LIN {X 64.801,Y 97.433,Z 77.000,A 180.000,B 0.000,C 180.000} C_DIS
LIN {X 64.718,Y 97.310,Z 77.000,A 180.000,B 0.000,C 180.000} C_DIS
LIN {X 64.539,Y 97.060,Z 77.000,A 180.000,B 0.000,C 180.000} C_DIS
LIN {X 64.421,Y 96.897,Z 77.000,A 180.000,B 0.000,C 180.000} C_DIS
LIN {X 64.360,Y 96.821,Z 77.000,A 180.000,B 0.000,C 180.000} C_DIS
LIN {X 64.272,Y 96.718,Z 77.000,A 180.000,B 0.000,C 180.000} C_DIS
LIN {X 64.119,Y 96.539,Z 77.000,A 180.000,B 0.000,C 180.000} C_DIS
LIN {X 64.003,Y 96.404,Z 77.000,A 180.000,B 0.000,C 180.000} C_DIS
LIN {X 63.962,Y 96.360,Z 77.000,A 180.000,B 0.000,C 180.000} C_DIS
LIN {X 63.824,Y 96.223,Z 77.000,A 180.000,B 0.000,C 180.000} C_DIS
LIN {X 63.599,Y 96.003,Z 77.000,A 180.000,B 0.000,C 180.000} C_DIS
LIN {X 63.467,Y 95.880,Z 77.000,A 180.000,B 0.000,C 180.000} C_DIS
LIN {X 63.399,Y 95.824,Z 77.000,A 180.000,B 0.000,C 180.000} C_DIS
LIN {X 63.109,Y 95.587,Z 77.000,A 180.000,B 0.000,C 180.000} C_DIS
LIN {X 62.954,Y 95.466,Z 77.000,A 180.000,B 0.000,C 180.000} C_DIS
LIN {X 62.930,Y 95.449,Z 77.000,A 180.000,B 0.000,C 180.000} C_DIS
LIN {X 62.751,Y 95.327,Z 77.000,A 180.000,B 0.000,C 180.000} C_DIS
LIN {X 62.573,Y 95.206,Z 77.000,A 180.000,B 0.000,C 180.000} C_DIS
LIN {X 62.425,Y 95.109,Z 77.000,A 180.000,B 0.000,C 180.000} C_DIS
LIN {X 62.394,Y 95.091,Z 77.000,A 180.000,B 0.000,C 180.000} C_DIS
LIN {X 62.215,Y 94.990,Z 77.000,A 180.000,B 0.000,C 180.000} C_DIS
LIN {X 62.036,Y 94.890,Z 77.000,A 180.000,B 0.000,C 180.000} C_DIS
LIN {X 61.858,Y 94.794,Z 77.000,A 180.000,B 0.000,C 180.000} C_DIS
LIN {X 61.769,Y 94.751,Z 77.000,A 180.000,B 0.000,C 180.000} C_DIS
LIN {X 61.679,Y 94.711,Z 77.000,A 180.000,B 0.000,C 180.000} C_DIS
LIN {X 61.369,Y 94.573,Z 77.000,A 180.000,B 0.000,C 180.000} C_DIS
LIN {X 61.321,Y 94.552,Z 77.000,A 180.000,B 0.000,C 180.000} C_DIS
LIN {X 61.143,Y 94.483,Z 77.000,A 180.000,B 0.000,C 180.000} C_DIS
LIN {X 60.785,Y 94.360,Z 77.000,A 180.000,B 0.000,C 180.000} C_DIS
LIN {X 60.606,Y 94.302,Z 77.000,A 180.000,B 0.000,C 180.000} C_DIS
LIN {X 60.427,Y 94.256,Z 77.000,A 180.000,B 0.000,C 180.000} C_DIS
LIN {X 60.249,Y 94.212,Z 77.000,A 180.000,B 0.000,C 180.000} C_DIS
LIN {X 60.070,Y 94.167,Z 77.000,A 180.000,B 0.000,C 180.000} C_DIS
LIN {X 59.891,Y 94.131,Z 77.000,A 180.000,B 0.000,C 180.000} C_DIS
LIN {X 59.712,Y 94.103,Z 77.000,A 180.000,B 0.000,C 180.000} C_DIS
LIN {X 59.534,Y 94.075,Z 77.000,A 180.000,B 0.000,C 180.000} C_DIS
LIN {X 59.355,Y 94.049,Z 77.000,A 180.000,B 0.000,C 180.000} C_DIS
LIN {X 59.220,Y 94.036,Z 77.000,A 180.000,B 0.000,C 180.000} C_DIS
LIN {X 58.819,Y 94.010,Z 77.000,A 180.000,B 0.000,C 180.000} C_DIS
LIN {X 58.640,Y 94.001,Z 77.000,A 180.000,B 0.000,C 180.000} C_DIS
LIN {X 58.461,Y 94.004,Z 77.000,A 180.000,B 0.000,C 180.000} C_DIS
LIN {X 58.282,Y 94.008,Z 77.000,A 180.000,B 0.000,C 180.000} C_DIS
LIN {X 58.103,Y 94.012,Z 77.000,A 180.000,B 0.000,C 180.000} C_DIS
LIN {X 57.925,Y 94.023,Z 77.000,A 180.000,B 0.000,C 180.000} C_DIS
LIN {X 57.803,Y 94.036,Z 77.000,A 180.000,B 0.000,C 180.000} C_DIS
LIN {X 57.567,Y 94.062,Z 77.000,A 180.000,B 0.000,C 180.000} C_DIS
LIN {X 57.388,Y 94.083,Z 77.000,A 180.000,B 0.000,C 180.000} C_DIS
LIN {X 57.210,Y 94.114,Z 77.000,A 180.000,B 0.000,C 180.000} C_DIS
LIN {X 56.852,Y 94.186,Z 77.000,A 180.000,B 0.000,C 180.000} C_DIS
LIN {X 56.717,Y 94.215,Z 77.000,A 180.000,B 0.000,C 180.000} C_DIS
LIN {X 56.673,Y 94.226,Z 77.000,A 180.000,B 0.000,C 180.000} C_DIS
LIN {X 56.495,Y 94.277,Z 77.000,A 180.000,B 0.000,C 180.000} C_DIS
LIN {X 56.316,Y 94.330,Z 77.000,A 180.000,B 0.000,C 180.000} C_DIS
LIN {X 56.137,Y 94.383,Z 77.000,A 180.000,B 0.000,C 180.000} C_DIS
LIN {X 56.103,Y 94.394,Z 77.000,A 180.000,B 0.000,C 180.000} C_DIS
LIN {X 55.958,Y 94.445,Z 77.000,A 180.000,B 0.000,C 180.000} C_DIS
LIN {X 55.601,Y 94.587,Z 77.000,A 180.000,B 0.000,C 180.000} C_DIS
LIN {X 55.422,Y 94.661,Z 77.000,A 180.000,B 0.000,C 180.000} C_DIS
LIN {X 55.243,Y 94.749,Z 77.000,A 180.000,B 0.000,C 180.000} C_DIS
LIN {X 55.064,Y 94.838,Z 77.000,A 180.000,B 0.000,C 180.000} C_DIS
LIN {X 54.886,Y 94.929,Z 77.000,A 180.000,B 0.000,C 180.000} C_DIS
LIN {X 54.883,Y 94.930,Z 77.000,A 180.000,B 0.000,C 180.000} C_DIS
LIN {X 54.707,Y 95.033,Z 77.000,A 180.000,B 0.000,C 180.000} C_DIS
LIN {X 54.528,Y 95.144,Z 77.000,A 180.000,B 0.000,C 180.000} C_DIS
LIN {X 54.349,Y 95.254,Z 77.000,A 180.000,B 0.000,C 180.000} C_DIS
LIN {X 54.298,Y 95.288,Z 77.000,A 180.000,B 0.000,C 180.000} C_DIS
LIN {X 54.171,Y 95.379,Z 77.000,A 180.000,B 0.000,C 180.000} C_DIS
LIN {X 53.992,Y 95.512,Z 77.000,A 180.000,B 0.000,C 180.000} C_DIS
LIN {X 53.814,Y 95.645,Z 77.000,A 180.000,B 0.000,C 180.000} C_DIS
LIN {X 53.813,Y 95.646,Z 77.000,A 180.000,B 0.000,C 180.000} C_DIS
LIN {X 53.634,Y 95.796,Z 77.000,A 180.000,B 0.000,C 180.000} C_DIS
LIN {X 53.404,Y 96.003,Z 77.000,A 180.000,B 0.000,C 180.000} C_DIS
LIN {X 53.277,Y 96.118,Z 77.000,A 180.000,B 0.000,C 180.000} C_DIS
LIN {X 53.213,Y 96.181,Z 77.000,A 180.000,B 0.000,C 180.000} C_DIS
LIN {X 53.098,Y 96.303,Z 77.000,A 180.000,B 0.000,C 180.000} C_DIS
LIN {X 52.877,Y 96.539,Z 77.000,A 180.000,B 0.000,C 180.000} C_DIS
LIN {X 52.740,Y 96.698,Z 77.000,A 180.000,B 0.000,C 180.000} C_DIS
LIN {X 52.725,Y 96.718,Z 77.000,A 180.000,B 0.000,C 180.000} C_DIS
LIN {X 52.562,Y 96.927,Z 77.000,A 180.000,B 0.000,C 180.000} C_DIS
LIN {X 52.446,Y 97.075,Z 77.000,A 180.000,B 0.000,C 180.000} C_DIS
LIN {X 52.383,Y 97.161,Z 77.000,A 180.000,B 0.000,C 180.000} C_DIS
LIN {X 52.320,Y 97.254,Z 77.000,A 180.000,B 0.000,C 180.000} C_DIS
LIN {X 52.088,Y 97.612,Z 77.000,A 180.000,B 0.000,C 180.000} C_DIS
LIN {X 52.025,Y 97.715,Z 77.000,A 180.000,B 0.000,C 180.000} C_DIS
LIN {X 51.983,Y 97.790,Z 77.000,A 180.000,B 0.000,C 180.000} C_DIS
LIN {X 51.889,Y 97.969,Z 77.000,A 180.000,B 0.000,C 180.000} C_DIS
LIN {X 51.794,Y 98.148,Z 77.000,A 180.000,B 0.000,C 180.000} C_DIS
LIN {X 51.705,Y 98.327,Z 77.000,A 180.000,B 0.000,C 180.000} C_DIS
LIN {X 51.668,Y 98.412,Z 77.000,A 180.000,B 0.000,C 180.000} C_DIS
LIN {X 51.553,Y 98.684,Z 77.000,A 180.000,B 0.000,C 180.000} C_DIS
LIN {X 51.489,Y 98.838,Z 77.000,A 180.000,B 0.000,C 180.000} C_DIS
LIN {X 51.479,Y 98.863,Z 77.000,A 180.000,B 0.000,C 180.000} C_DIS
LIN {X 51.417,Y 99.042,Z 77.000,A 180.000,B 0.000,C 180.000} C_DIS
LIN {X 51.303,Y 99.399,Z 77.000,A 180.000,B 0.000,C 180.000} C_DIS
LIN {X 51.251,Y 99.578,Z 77.000,A 180.000,B 0.000,C 180.000} C_DIS
LIN {X 51.210,Y 99.757,Z 77.000,A 180.000,B 0.000,C 180.000} C_DIS
LIN {X 51.170,Y 99.936,Z 77.000,A 180.000,B 0.000,C 180.000} C_DIS
LIN {X 51.131,Y 100.106,Z 77.000,A 180.000,B 0.000,C 180.000} C_DIS
LIN {X 51.130,Y 100.114,Z 77.000,A 180.000,B 0.000,C 180.000} C_DIS
LIN {X 51.100,Y 100.293,Z 77.000,A 180.000,B 0.000,C 180.000} C_DIS
LIN {X 51.052,Y 100.651,Z 77.000,A 180.000,B 0.000,C 180.000} C_DIS
LIN {X 51.030,Y 100.829,Z 77.000,A 180.000,B 0.000,C 180.000} C_DIS
LIN {X 51.019,Y 101.008,Z 77.000,A 180.000,B 0.000,C 180.000} C_DIS
LIN {X 51.003,Y 101.366,Z 77.000,A 180.000,B 0.000,C 180.000} C_DIS
LIN {X 51.000,Y 101.545,Z 77.000,A 180.000,B 0.000,C 180.000} C_DIS
LIN {X 51.007,Y 101.723,Z 77.000,A 180.000,B 0.000,C 180.000} C_DIS
LIN {X 51.015,Y 101.902,Z 77.000,A 180.000,B 0.000,C 180.000} C_DIS
LIN {X 51.023,Y 102.081,Z 77.000,A 180.000,B 0.000,C 180.000} C_DIS
LIN {X 51.040,Y 102.260,Z 77.000,A 180.000,B 0.000,C 180.000} C_DIS
LIN {X 51.064,Y 102.438,Z 77.000,A 180.000,B 0.000,C 180.000} C_DIS
LIN {X 51.088,Y 102.617,Z 77.000,A 180.000,B 0.000,C 180.000} C_DIS
LIN {X 51.113,Y 102.796,Z 77.000,A 180.000,B 0.000,C 180.000} C_DIS
LIN {X 51.131,Y 102.894,Z 77.000,A 180.000,B 0.000,C 180.000} C_DIS
LIN {X 51.149,Y 102.975,Z 77.000,A 180.000,B 0.000,C 180.000} C_DIS
LIN {X 51.230,Y 103.332,Z 77.000,A 180.000,B 0.000,C 180.000} C_DIS
LIN {X 51.275,Y 103.511,Z 77.000,A 180.000,B 0.000,C 180.000} C_DIS
LIN {X 51.310,Y 103.624,Z 77.000,A 180.000,B 0.000,C 180.000} C_DIS
LIN {X 51.388,Y 103.869,Z 77.000,A 180.000,B 0.000,C 180.000} C_DIS
LIN {X 51.446,Y 104.047,Z 77.000,A 180.000,B 0.000,C 180.000} C_DIS
LIN {X 51.489,Y 104.162,Z 77.000,A 180.000,B 0.000,C 180.000} C_DIS
LIN {X 51.515,Y 104.226,Z 77.000,A 180.000,B 0.000,C 180.000} C_DIS
LIN {X 51.668,Y 104.588,Z 77.000,A 180.000,B 0.000,C 180.000} C_DIS
LIN {X 51.747,Y 104.762,Z 77.000,A 180.000,B 0.000,C 180.000} C_DIS
LIN {X 51.841,Y 104.941,Z 77.000,A 180.000,B 0.000,C 180.000} C_DIS
LIN {X 51.936,Y 105.120,Z 77.000,A 180.000,B 0.000,C 180.000} C_DIS
LIN {X 52.025,Y 105.285,Z 77.000,A 180.000,B 0.000,C 180.000} C_DIS
LIN {X 52.033,Y 105.299,Z 77.000,A 180.000,B 0.000,C 180.000} C_DIS
LIN {X 52.146,Y 105.477,Z 77.000,A 180.000,B 0.000,C 180.000} C_DIS
LIN {X 52.262,Y 105.656,Z 77.000,A 180.000,B 0.000,C 180.000} C_DIS
LIN {X 52.380,Y 105.835,Z 77.000,A 180.000,B 0.000,C 180.000} C_DIS
LIN {X 52.383,Y 105.839,Z 77.000,A 180.000,B 0.000,C 180.000} C_DIS
LIN {X 52.515,Y 106.014,Z 77.000,A 180.000,B 0.000,C 180.000} C_DIS
LIN {X 52.655,Y 106.193,Z 77.000,A 180.000,B 0.000,C 180.000} C_DIS
LIN {X 52.740,Y 106.302,Z 77.000,A 180.000,B 0.000,C 180.000} C_DIS
LIN {X 52.797,Y 106.371,Z 77.000,A 180.000,B 0.000,C 180.000} C_DIS
LIN {X 52.919,Y 106.506,Z 77.000,A 180.000,B 0.000,C 180.000} C_DIS
LIN {X 53.128,Y 106.729,Z 77.000,A 180.000,B 0.000,C 180.000} C_DIS
LIN {X 53.277,Y 106.882,Z 77.000,A 180.000,B 0.000,C 180.000} C_DIS
LIN {X 53.304,Y 106.908,Z 77.000,A 180.000,B 0.000,C 180.000} C_DIS
LIN {X 53.455,Y 107.044,Z 77.000,A 180.000,B 0.000,C 180.000} C_DIS
LIN {X 53.634,Y 107.204,Z 77.000,A 180.000,B 0.000,C 180.000} C_DIS
LIN {X 53.704,Y 107.265,Z 77.000,A 180.000,B 0.000,C 180.000} C_DIS
LIN {X 53.813,Y 107.354,Z 77.000,A 180.000,B 0.000,C 180.000} C_DIS
LIN {X 53.933,Y 107.444,Z 77.000,A 180.000,B 0.000,C 180.000} C_DIS
LIN {X 54.172,Y 107.623,Z 77.000,A 180.000,B 0.000,C 180.000} C_DIS
LIN {X 54.349,Y 107.746,Z 77.000,A 180.000,B 0.000,C 180.000} C_DIS
LIN {X 54.439,Y 107.802,Z 77.000,A 180.000,B 0.000,C 180.000} C_DIS
LIN {X 54.729,Y 107.980,Z 77.000,A 180.000,B 0.000,C 180.000} C_DIS
LIN {X 54.886,Y 108.071,Z 77.000,A 180.000,B 0.000,C 180.000} C_DIS
LIN {X 55.059,Y 108.159,Z 77.000,A 180.000,B 0.000,C 180.000} C_DIS
LIN {X 55.243,Y 108.251,Z 77.000,A 180.000,B 0.000,C 180.000} C_DIS
LIN {X 55.419,Y 108.338,Z 77.000,A 180.000,B 0.000,C 180.000} C_DIS
LIN {X 55.422,Y 108.339,Z 77.000,A 180.000,B 0.000,C 180.000} C_DIS
LIN {X 55.601,Y 108.413,Z 77.000,A 180.000,B 0.000,C 180.000} C_DIS
LIN {X 55.862,Y 108.517,Z 77.000,A 180.000,B 0.000,C 180.000} C_DIS
LIN {X 55.958,Y 108.555,Z 77.000,A 180.000,B 0.000,C 180.000} C_DIS
LIN {X 56.137,Y 108.617,Z 77.000,A 180.000,B 0.000,C 180.000} C_DIS
LIN {X 56.316,Y 108.670,Z 77.000,A 180.000,B 0.000,C 180.000} C_DIS
LIN {X 56.495,Y 108.723,Z 77.000,A 180.000,B 0.000,C 180.000} C_DIS
LIN {X 56.673,Y 108.774,Z 77.000,A 180.000,B 0.000,C 180.000} C_DIS
LIN {X 56.852,Y 108.814,Z 77.000,A 180.000,B 0.000,C 180.000} C_DIS
LIN {X 57.210,Y 108.886,Z 77.000,A 180.000,B 0.000,C 180.000} C_DIS
LIN {X 57.388,Y 108.917,Z 77.000,A 180.000,B 0.000,C 180.000} C_DIS
LIN {X 57.567,Y 108.938,Z 77.000,A 180.000,B 0.000,C 180.000} C_DIS
LIN {X 57.746,Y 108.957,Z 77.000,A 180.000,B 0.000,C 180.000} C_DIS
LIN {X 57.925,Y 108.977,Z 77.000,A 180.000,B 0.000,C 180.000} C_DIS
LIN {X 58.103,Y 108.988,Z 77.000,A 180.000,B 0.000,C 180.000} C_DIS
LIN {X 58.282,Y 108.992,Z 77.000,A 180.000,B 0.000,C 180.000} C_DIS
LIN {X 58.461,Y 108.996,Z 77.000,A 180.000,B 0.000,C 180.000} C_DIS
LIN {X 58.640,Y 108.999,Z 77.000,A 180.000,B 0.000,C 180.000} C_DIS
LIN {X 58.819,Y 108.990,Z 77.000,A 180.000,B 0.000,C 180.000} C_DIS
LIN {X 59.176,Y 108.967,Z 77.000,A 180.000,B 0.000,C 180.000} C_DIS
LIN {X 59.355,Y 108.951,Z 77.000,A 180.000,B 0.000,C 180.000} C_DIS
LIN {X 59.534,Y 108.925,Z 77.000,A 180.000,B 0.000,C 180.000} C_DIS
LIN {X 59.856,Y 108.874,Z 77.000,A 180.000,B 0.000,C 180.000} C_DIS
LIN {X 59.891,Y 108.869,Z 77.000,A 180.000,B 0.000,C 180.000} C_DIS
LIN {X 60.070,Y 108.833,Z 77.000,A 180.000,B 0.000,C 180.000} C_DIS
LIN {X 60.249,Y 108.788,Z 77.000,A 180.000,B 0.000,C 180.000} C_DIS
LIN {X 60.427,Y 108.744,Z 77.000,A 180.000,B 0.000,C 180.000} C_DIS
LIN {X 60.606,Y 108.698,Z 77.000,A 180.000,B 0.000,C 180.000} C_DIS
LIN {X 60.616,Y 108.695,Z 77.000,A 180.000,B 0.000,C 180.000} C_DIS
LIN {X 60.785,Y 108.640,Z 77.000,A 180.000,B 0.000,C 180.000} C_DIS
LIN {X 61.144,Y 108.517,Z 77.000,A 180.000,B 0.000,C 180.000} C_DIS
LIN {X 61.321,Y 108.448,Z 77.000,A 180.000,B 0.000,C 180.000} C_DIS
LIN {X 61.500,Y 108.369,Z 77.000,A 180.000,B 0.000,C 180.000} C_DIS
LIN {X 61.679,Y 108.289,Z 77.000,A 180.000,B 0.000,C 180.000} C_DIS
LIN {X 61.858,Y 108.206,Z 77.000,A 180.000,B 0.000,C 180.000} C_DIS
LIN {X 61.948,Y 108.159,Z 77.000,A 180.000,B 0.000,C 180.000} C_DIS
LIN {X 62.036,Y 108.110,Z 77.000,A 180.000,B 0.000,C 180.000} C_DIS
LIN {X 62.268,Y 107.980,Z 77.000,A 180.000,B 0.000,C 180.000} C_DIS
LIN {X 62.394,Y 107.909,Z 77.000,A 180.000,B 0.000,C 180.000} C_DIS
LIN {X 62.562,Y 107.802,Z 77.000,A 180.000,B 0.000,C 180.000} C_DIS
LIN {X 62.825,Y 107.623,Z 77.000,A 180.000,B 0.000,C 180.000} C_DIS
LIN {X 62.930,Y 107.551,Z 77.000,A 180.000,B 0.000,C 180.000} C_DIS
LIN {X 63.071,Y 107.444,Z 77.000,A 180.000,B 0.000,C 180.000} C_DIS
LIN {X 63.109,Y 107.413,Z 77.000,A 180.000,B 0.000,C 180.000} C_DIS
LIN {X 63.290,Y 107.265,Z 77.000,A 180.000,B 0.000,C 180.000} C_DIS
LIN {X 63.467,Y 107.120,Z 77.000,A 180.000,B 0.000,C 180.000} C_DIS
LIN {X 63.504,Y 107.086,Z 77.000,A 180.000,B 0.000,C 180.000} C_DIS
LIN {X 63.645,Y 106.952,Z 77.000,A 180.000,B 0.000,C 180.000} C_DIS
LIN {X 63.873,Y 106.729,Z 77.000,A 180.000,B 0.000,C 180.000} C_DIS
LIN {X 64.003,Y 106.596,Z 77.000,A 180.000,B 0.000,C 180.000} C_DIS
LIN {X 64.043,Y 106.550,Z 77.000,A 180.000,B 0.000,C 180.000} C_DIS
LIN {X 64.196,Y 106.371,Z 77.000,A 180.000,B 0.000,C 180.000} C_DIS
LIN {X 64.349,Y 106.193,Z 77.000,A 180.000,B 0.000,C 180.000} C_DIS
LIN {X 64.360,Y 106.179,Z 77.000,A 180.000,B 0.000,C 180.000} C_DIS
LIN {X 64.487,Y 106.014,Z 77.000,A 180.000,B 0.000,C 180.000} C_DIS
LIN {X 64.718,Y 105.690,Z 77.000,A 180.000,B 0.000,C 180.000} C_DIS
LIN {X 64.742,Y 105.656,Z 77.000,A 180.000,B 0.000,C 180.000} C_DIS
LIN {X 64.856,Y 105.477,Z 77.000,A 180.000,B 0.000,C 180.000} C_DIS
LIN {X 65.075,Y 105.104,Z 77.000,A 180.000,B 0.000,C 180.000} C_DIS
LIN {X 65.163,Y 104.941,Z 77.000,A 180.000,B 0.000,C 180.000} C_DIS
LIN {X 65.248,Y 104.762,Z 77.000,A 180.000,B 0.000,C 180.000} C_DIS
LIN {X 65.333,Y 104.584,Z 77.000,A 180.000,B 0.000,C 180.000} C_DIS
LIN {X 65.415,Y 104.405,Z 77.000,A 180.000,B 0.000,C 180.000} C_DIS
LIN {X 65.433,Y 104.360,Z 77.000,A 180.000,B 0.000,C 180.000} C_DIS
LIN {X 65.483,Y 104.226,Z 77.000,A 180.000,B 0.000,C 180.000} C_DIS
LIN {X 65.549,Y 104.047,Z 77.000,A 180.000,B 0.000,C 180.000} C_DIS
LIN {X 65.612,Y 103.878,Z 77.000,A 180.000,B 0.000,C 180.000} C_DIS
LIN {X 65.615,Y 103.869,Z 77.000,A 180.000,B 0.000,C 180.000} C_DIS
LIN {X 65.672,Y 103.690,Z 77.000,A 180.000,B 0.000,C 180.000} C_DIS
LIN {X 65.720,Y 103.511,Z 77.000,A 180.000,B 0.000,C 180.000} C_DIS
LIN {X 65.791,Y 103.253,Z 77.000,A 180.000,B 0.000,C 180.000} C_DIS
LIN {X 65.815,Y 103.153,Z 77.000,A 180.000,B 0.000,C 180.000} C_DIS
LIN {X 65.850,Y 102.975,Z 77.000,A 180.000,B 0.000,C 180.000} C_DIS
LIN {X 65.914,Y 102.617,Z 77.000,A 180.000,B 0.000,C 180.000} C_DIS
LIN {X 65.941,Y 102.438,Z 77.000,A 180.000,B 0.000,C 180.000} C_DIS
LIN {X 65.957,Y 102.260,Z 77.000,A 180.000,B 0.000,C 180.000} C_DIS
LIN {X 65.973,Y 102.081,Z 77.000,A 180.000,B 0.000,C 180.000} C_DIS
LIN {X 65.989,Y 101.902,Z 77.000,A 180.000,B 0.000,C 180.000} C_DIS
LIN {X 65.995,Y 101.723,Z 77.000,A 180.000,B 0.000,C 180.000} C_DIS
LIN {X 65.995,Y 101.366,Z 77.000,A 180.000,B 0.000,C 180.000} C_DIS
LIN {X 65.993,Y 101.187,Z 77.000,A 180.000,B 0.000,C 180.000} C_DIS
LIN {X 65.981,Y 101.008,Z 77.000,A 180.000,B 0.000,C 180.000} C_DIS
LIN {X 65.949,Y 100.651,Z 77.000,A 180.000,B 0.000,C 180.000} C_DIS
LIN {X 65.929,Y 100.472,Z 77.000,A 180.000,B 0.000,C 180.000} C_DIS
LIN {X 65.898,Y 100.293,Z 77.000,A 180.000,B 0.000,C 180.000} C_DIS
LIN {X 65.866,Y 100.114,Z 77.000,A 180.000,B 0.000,C 180.000} C_DIS
LIN {X 65.834,Y 99.936,Z 77.000,A 180.000,B 0.000,C 180.000} C_DIS
LIN {X 65.793,Y 99.757,Z 77.000,A 180.000,B 0.000,C 180.000} C_DIS
LIN {X 65.791,Y 99.747,Z 77.000,A 180.000,B 0.000,C 180.000} C_DIS
LIN {X 65.696,Y 99.399,Z 77.000,A 180.000,B 0.000,C 180.000} C_DIS
LIN {X 65.645,Y 99.221,Z 77.000,A 180.000,B 0.000,C 180.000} C_DIS
LIN {X 65.612,Y 99.122,Z 77.000,A 180.000,B 0.000,C 180.000} C_DIS
; Link Move Starts
LIN {X 65.503,Y 98.827,Z 77.000,A 180.000,B 0.000,C 180.000} C_DIS
LIN {X 65.388,Y 98.534,Z 76.999,A 180.000,B 0.000,C 180.000} C_DIS
LIN {X 65.253,Y 98.249,Z 76.998,A 180.000,B 0.000,C 180.000} C_DIS
LIN {X 65.115,Y 97.966,Z 76.996,A 180.000,B 0.000,C 180.000} C_DIS
LIN {X 64.957,Y 97.693,Z 76.994,A 180.000,B 0.000,C 180.000} C_DIS
LIN {X 64.795,Y 97.423,Z 76.991,A 180.000,B 0.000,C 180.000} C_DIS
LIN {X 64.614,Y 97.165,Z 76.988,A 180.000,B 0.000,C 180.000} C_DIS
LIN {X 64.431,Y 96.909,Z 76.985,A 180.000,B 0.000,C 180.000} C_DIS
LIN {X 64.229,Y 96.667,Z 76.981,A 180.000,B 0.000,C 180.000} C_DIS
LIN {X 64.024,Y 96.428,Z 76.977,A 180.000,B 0.000,C 180.000} C_DIS
LIN {X 63.804,Y 96.203,Z 76.972,A 180.000,B 0.000,C 180.000} C_DIS
LIN {X 63.691,Y 96.093,Z 76.969,A 180.000,B 0.000,C 180.000} C_DIS
LIN {X 63.578,Y 95.983,Z 76.967,A 180.000,B 0.000,C 180.000} C_DIS
LIN {X 63.462,Y 95.877,Z 76.964,A 180.000,B 0.000,C 180.000} C_DIS
LIN {X 63.341,Y 95.776,Z 76.961,A 180.000,B 0.000,C 180.000} C_DIS
LIN {X 63.219,Y 95.677,Z 76.959,A 180.000,B 0.000,C 180.000} C_DIS
LIN {X 63.097,Y 95.577,Z 76.956,A 180.000,B 0.000,C 180.000} C_DIS
LIN {X 62.973,Y 95.480,Z 76.952,A 180.000,B 0.000,C 180.000} C_DIS
LIN {X 62.844,Y 95.390,Z 76.949,A 180.000,B 0.000,C 180.000} C_DIS
LIN {X 62.713,Y 95.301,Z 76.946,A 180.000,B 0.000,C 180.000} C_DIS
LIN {X 62.583,Y 95.213,Z 76.943,A 180.000,B 0.000,C 180.000} C_DIS
LIN {X 62.452,Y 95.126,Z 76.939,A 180.000,B 0.000,C 180.000} C_DIS
LIN {X 62.316,Y 95.046,Z 76.936,A 180.000,B 0.000,C 180.000} C_DIS
LIN {X 62.178,Y 94.969,Z 76.932,A 180.000,B 0.000,C 180.000} C_DIS
LIN {X 62.041,Y 94.893,Z 76.928,A 180.000,B 0.000,C 180.000} C_DIS
LIN {X 61.903,Y 94.817,Z 76.925,A 180.000,B 0.000,C 180.000} C_DIS
LIN {X 61.761,Y 94.748,Z 76.921,A 180.000,B 0.000,C 180.000} C_DIS
LIN {X 61.617,Y 94.684,Z 76.917,A 180.000,B 0.000,C 180.000} C_DIS
LIN {X 61.474,Y 94.619,Z 76.913,A 180.000,B 0.000,C 180.000} C_DIS
LIN {X 61.330,Y 94.555,Z 76.909,A 180.000,B 0.000,C 180.000} C_DIS
LIN {X 61.183,Y 94.497,Z 76.905,A 180.000,B 0.000,C 180.000} C_DIS
LIN {X 61.034,Y 94.446,Z 76.900,A 180.000,B 0.000,C 180.000} C_DIS
LIN {X 60.885,Y 94.394,Z 76.896,A 180.000,B 0.000,C 180.000} C_DIS
LIN {X 60.737,Y 94.343,Z 76.892,A 180.000,B 0.000,C 180.000} C_DIS
LIN {X 60.586,Y 94.296,Z 76.887,A 180.000,B 0.000,C 180.000} C_DIS
LIN {X 60.434,Y 94.257,Z 76.883,A 180.000,B 0.000,C 180.000} C_DIS
LIN {X 60.281,Y 94.219,Z 76.878,A 180.000,B 0.000,C 180.000} C_DIS
LIN {X 60.128,Y 94.182,Z 76.873,A 180.000,B 0.000,C 180.000} C_DIS
LIN {X 59.974,Y 94.146,Z 76.869,A 180.000,B 0.000,C 180.000} C_DIS
LIN {X 59.819,Y 94.120,Z 76.864,A 180.000,B 0.000,C 180.000} C_DIS
LIN {X 59.663,Y 94.096,Z 76.859,A 180.000,B 0.000,C 180.000} C_DIS
LIN {X 59.508,Y 94.071,Z 76.854,A 180.000,B 0.000,C 180.000} C_DIS
LIN {X 59.430,Y 94.059,Z 76.851,A 180.000,B 0.000,C 180.000} C_DIS
LIN {X 59.352,Y 94.049,Z 76.849,A 180.000,B 0.000,C 180.000} C_DIS
LIN {X 59.274,Y 94.040,Z 76.846,A 180.000,B 0.000,C 180.000} C_DIS
LIN {X 59.195,Y 94.035,Z 76.844,A 180.000,B 0.000,C 180.000} C_DIS
LIN {X 59.117,Y 94.029,Z 76.841,A 180.000,B 0.000,C 180.000} C_DIS
LIN {X 59.038,Y 94.024,Z 76.839,A 180.000,B 0.000,C 180.000} C_DIS
LIN {X 58.959,Y 94.019,Z 76.836,A 180.000,B 0.000,C 180.000} C_DIS
LIN {X 58.802,Y 94.008,Z 76.831,A 180.000,B 0.000,C 180.000} C_DIS
LIN {X 58.724,Y 94.004,Z 76.828,A 180.000,B 0.000,C 180.000} C_DIS
LIN {X 58.645,Y 94.001,Z 76.825,A 180.000,B 0.000,C 180.000} C_DIS
LIN {X 58.566,Y 94.002,Z 76.823,A 180.000,B 0.000,C 180.000} C_DIS
LIN {X 58.487,Y 94.003,Z 76.820,A 180.000,B 0.000,C 180.000} C_DIS
LIN {X 58.330,Y 94.007,Z 76.815,A 180.000,B 0.000,C 180.000} C_DIS
LIN {X 58.172,Y 94.010,Z 76.809,A 180.000,B 0.000,C 180.000} C_DIS
LIN {X 58.094,Y 94.012,Z 76.807,A 180.000,B 0.000,C 180.000} C_DIS
LIN {X 58.015,Y 94.016,Z 76.804,A 180.000,B 0.000,C 180.000} C_DIS
LIN {X 57.937,Y 94.022,Z 76.801,A 180.000,B 0.000,C 180.000} C_DIS
LIN {X 57.858,Y 94.030,Z 76.798,A 180.000,B 0.000,C 180.000} C_DIS
LIN {X 57.780,Y 94.039,Z 76.796,A 180.000,B 0.000,C 180.000} C_DIS
LIN {X 57.623,Y 94.056,Z 76.790,A 180.000,B 0.000,C 180.000} C_DIS
LIN {X 57.467,Y 94.074,Z 76.785,A 180.000,B 0.000,C 180.000} C_DIS
LIN {X 57.389,Y 94.083,Z 76.782,A 180.000,B 0.000,C 180.000} C_DIS
LIN {X 57.311,Y 94.095,Z 76.779,A 180.000,B 0.000,C 180.000} C_DIS
LIN {X 57.233,Y 94.109,Z 76.776,A 180.000,B 0.000,C 180.000} C_DIS
LIN {X 57.156,Y 94.125,Z 76.774,A 180.000,B 0.000,C 180.000} C_DIS
LIN {X 57.002,Y 94.156,Z 76.768,A 180.000,B 0.000,C 180.000} C_DIS
LIN {X 56.847,Y 94.187,Z 76.763,A 180.000,B 0.000,C 180.000} C_DIS
LIN {X 56.770,Y 94.203,Z 76.760,A 180.000,B 0.000,C 180.000} C_DIS
LIN {X 56.694,Y 94.221,Z 76.757,A 180.000,B 0.000,C 180.000} C_DIS
LIN {X 56.617,Y 94.241,Z 76.754,A 180.000,B 0.000,C 180.000} C_DIS
LIN {X 56.542,Y 94.263,Z 76.752,A 180.000,B 0.000,C 180.000} C_DIS
LIN {X 56.391,Y 94.308,Z 76.746,A 180.000,B 0.000,C 180.000} C_DIS
LIN {X 56.164,Y 94.375,Z 76.738,A 180.000,B 0.000,C 180.000} C_DIS
LIN {X 56.089,Y 94.398,Z 76.735,A 180.000,B 0.000,C 180.000} C_DIS
LIN {X 56.015,Y 94.424,Z 76.732,A 180.000,B 0.000,C 180.000} C_DIS
LIN {X 55.941,Y 94.452,Z 76.730,A 180.000,B 0.000,C 180.000} C_DIS
LIN {X 55.795,Y 94.510,Z 76.724,A 180.000,B 0.000,C 180.000} C_DIS
LIN {X 55.575,Y 94.597,Z 76.716,A 180.000,B 0.000,C 180.000} C_DIS
LIN {X 55.502,Y 94.626,Z 76.713,A 180.000,B 0.000,C 180.000} C_DIS
LIN {X 55.429,Y 94.657,Z 76.710,A 180.000,B 0.000,C 180.000} C_DIS
LIN {X 55.358,Y 94.691,Z 76.708,A 180.000,B 0.000,C 180.000} C_DIS
LIN {X 55.288,Y 94.726,Z 76.705,A 180.000,B 0.000,C 180.000} C_DIS
LIN {X 55.147,Y 94.797,Z 76.699,A 180.000,B 0.000,C 180.000} C_DIS
LIN {X 55.077,Y 94.832,Z 76.697,A 180.000,B 0.000,C 180.000} C_DIS
LIN {X 55.006,Y 94.867,Z 76.694,A 180.000,B 0.000,C 180.000} C_DIS
LIN {X 54.936,Y 94.903,Z 76.691,A 180.000,B 0.000,C 180.000} C_DIS
LIN {X 54.866,Y 94.939,Z 76.688,A 180.000,B 0.000,C 180.000} C_DIS
LIN {X 54.798,Y 94.978,Z 76.686,A 180.000,B 0.000,C 180.000} C_DIS
LIN {X 54.730,Y 95.019,Z 76.683,A 180.000,B 0.000,C 180.000} C_DIS
LIN {X 54.596,Y 95.102,Z 76.677,A 180.000,B 0.000,C 180.000} C_DIS
LIN {X 54.529,Y 95.143,Z 76.675,A 180.000,B 0.000,C 180.000} C_DIS
LIN {X 54.395,Y 95.226,Z 76.669,A 180.000,B 0.000,C 180.000} C_DIS
LIN {X 54.328,Y 95.268,Z 76.666,A 180.000,B 0.000,C 180.000} C_DIS
LIN {X 54.263,Y 95.312,Z 76.664,A 180.000,B 0.000,C 180.000} C_DIS
LIN {X 54.199,Y 95.357,Z 76.661,A 180.000,B 0.000,C 180.000} C_DIS
LIN {X 54.136,Y 95.405,Z 76.658,A 180.000,B 0.000,C 180.000} C_DIS
LIN {X 53.884,Y 95.593,Z 76.647,A 180.000,B 0.000,C 180.000} C_DIS
LIN {X 53.821,Y 95.640,Z 76.644,A 180.000,B 0.000,C 180.000} C_DIS
LIN {X 53.759,Y 95.689,Z 76.642,A 180.000,B 0.000,C 180.000} C_DIS
LIN {X 53.698,Y 95.739,Z 76.639,A 180.000,B 0.000,C 180.000} C_DIS
LIN {X 53.639,Y 95.792,Z 76.636,A 180.000,B 0.000,C 180.000} C_DIS
LIN {X 53.346,Y 96.054,Z 76.622,A 180.000,B 0.000,C 180.000} C_DIS
LIN {X 53.288,Y 96.107,Z 76.620,A 180.000,B 0.000,C 180.000} C_DIS
LIN {X 53.231,Y 96.162,Z 76.617,A 180.000,B 0.000,C 180.000} C_DIS
LIN {X 53.177,Y 96.219,Z 76.614,A 180.000,B 0.000,C 180.000} C_DIS
LIN {X 52.908,Y 96.507,Z 76.600,A 180.000,B 0.000,C 180.000} C_DIS
LIN {X 52.854,Y 96.564,Z 76.598,A 180.000,B 0.000,C 180.000} C_DIS
LIN {X 52.802,Y 96.623,Z 76.595,A 180.000,B 0.000,C 180.000} C_DIS
LIN {X 52.752,Y 96.684,Z 76.592,A 180.000,B 0.000,C 180.000} C_DIS
LIN {X 52.703,Y 96.746,Z 76.589,A 180.000,B 0.000,C 180.000} C_DIS
LIN {X 52.460,Y 97.056,Z 76.576,A 180.000,B 0.000,C 180.000} C_DIS
LIN {X 52.413,Y 97.119,Z 76.573,A 180.000,B 0.000,C 180.000} C_DIS
LIN {X 52.367,Y 97.183,Z 76.570,A 180.000,B 0.000,C 180.000} C_DIS
LIN {X 52.324,Y 97.249,Z 76.567,A 180.000,B 0.000,C 180.000} C_DIS
LIN {X 52.110,Y 97.579,Z 76.554,A 180.000,B 0.000,C 180.000} C_DIS
LIN {X 52.067,Y 97.645,Z 76.551,A 180.000,B 0.000,C 180.000} C_DIS
LIN {X 52.026,Y 97.713,Z 76.548,A 180.000,B 0.000,C 180.000} C_DIS
LIN {X 51.988,Y 97.782,Z 76.545,A 180.000,B 0.000,C 180.000} C_DIS
LIN {X 51.951,Y 97.851,Z 76.543,A 180.000,B 0.000,C 180.000} C_DIS
LIN {X 51.804,Y 98.130,Z 76.532,A 180.000,B 0.000,C 180.000} C_DIS
LIN {X 51.767,Y 98.199,Z 76.529,A 180.000,B 0.000,C 180.000} C_DIS
LIN {X 51.731,Y 98.270,Z 76.526,A 180.000,B 0.000,C 180.000} C_DIS
LIN {X 51.698,Y 98.341,Z 76.523,A 180.000,B 0.000,C 180.000} C_DIS
LIN {X 51.667,Y 98.413,Z 76.521,A 180.000,B 0.000,C 180.000} C_DIS
LIN {X 51.515,Y 98.776,Z 76.507,A 180.000,B 0.000,C 180.000} C_DIS
LIN {X 51.485,Y 98.849,Z 76.504,A 180.000,B 0.000,C 180.000} C_DIS
LIN {X 51.457,Y 98.923,Z 76.501,A 180.000,B 0.000,C 180.000} C_DIS
LIN {X 51.431,Y 98.997,Z 76.499,A 180.000,B 0.000,C 180.000} C_DIS
LIN {X 51.383,Y 99.147,Z 76.493,A 180.000,B 0.000,C 180.000} C_DIS
LIN {X 51.311,Y 99.372,Z 76.485,A 180.000,B 0.000,C 180.000} C_DIS
LIN {X 51.287,Y 99.447,Z 76.482,A 180.000,B 0.000,C 180.000} C_DIS
LIN {X 51.265,Y 99.523,Z 76.479,A 180.000,B 0.000,C 180.000} C_DIS
LIN {X 51.246,Y 99.599,Z 76.477,A 180.000,B 0.000,C 180.000} C_DIS
LIN {X 51.228,Y 99.676,Z 76.474,A 180.000,B 0.000,C 180.000} C_DIS
LIN {X 51.142,Y 100.060,Z 76.460,A 180.000,B 0.000,C 180.000} C_DIS
LIN {X 51.125,Y 100.137,Z 76.457,A 180.000,B 0.000,C 180.000} C_DIS
LIN {X 51.111,Y 100.215,Z 76.455,A 180.000,B 0.000,C 180.000} C_DIS
LIN {X 51.100,Y 100.293,Z 76.452,A 180.000,B 0.000,C 180.000} C_DIS
LIN {X 51.047,Y 100.683,Z 76.438,A 180.000,B 0.000,C 180.000} C_DIS
LIN {X 51.037,Y 100.761,Z 76.435,A 180.000,B 0.000,C 180.000} C_DIS
LIN {X 51.029,Y 100.839,Z 76.433,A 180.000,B 0.000,C 180.000} C_DIS
LIN {X 51.024,Y 100.918,Z 76.430,A 180.000,B 0.000,C 180.000} C_DIS
LIN {X 51.020,Y 100.997,Z 76.427,A 180.000,B 0.000,C 180.000} C_DIS
LIN {X 51.002,Y 101.390,Z 76.413,A 180.000,B 0.000,C 180.000} C_DIS
LIN {X 51.000,Y 101.469,Z 76.411,A 180.000,B 0.000,C 180.000} C_DIS
LIN {X 51.000,Y 101.547,Z 76.408,A 180.000,B 0.000,C 180.000} C_DIS
LIN {X 51.003,Y 101.626,Z 76.405,A 180.000,B 0.000,C 180.000} C_DIS
LIN {X 51.021,Y 102.019,Z 76.391,A 180.000,B 0.000,C 180.000} C_DIS
LIN {X 51.024,Y 102.098,Z 76.389,A 180.000,B 0.000,C 180.000} C_DIS
LIN {X 51.031,Y 102.177,Z 76.386,A 180.000,B 0.000,C 180.000} C_DIS
LIN {X 51.039,Y 102.255,Z 76.383,A 180.000,B 0.000,C 180.000} C_DIS
LIN {X 51.050,Y 102.333,Z 76.380,A 180.000,B 0.000,C 180.000} C_DIS
LIN {X 51.070,Y 102.489,Z 76.375,A 180.000,B 0.000,C 180.000} C_DIS
LIN {X 51.091,Y 102.645,Z 76.369,A 180.000,B 0.000,C 180.000} C_DIS
LIN {X 51.102,Y 102.723,Z 76.367,A 180.000,B 0.000,C 180.000} C_DIS
LIN {X 51.114,Y 102.801,Z 76.364,A 180.000,B 0.000,C 180.000} C_DIS
LIN {X 51.128,Y 102.879,Z 76.361,A 180.000,B 0.000,C 180.000} C_DIS
LIN {X 51.145,Y 102.955,Z 76.358,A 180.000,B 0.000,C 180.000} C_DIS
LIN {X 51.180,Y 103.109,Z 76.353,A 180.000,B 0.000,C 180.000} C_DIS
LIN {X 51.231,Y 103.340,Z 76.345,A 180.000,B 0.000,C 180.000} C_DIS
LIN {X 51.249,Y 103.416,Z 76.342,A 180.000,B 0.000,C 180.000} C_DIS
LIN {X 51.270,Y 103.492,Z 76.339,A 180.000,B 0.000,C 180.000} C_DIS
LIN {X 51.292,Y 103.568,Z 76.336,A 180.000,B 0.000,C 180.000} C_DIS
LIN {X 51.316,Y 103.643,Z 76.334,A 180.000,B 0.000,C 180.000} C_DIS
LIN {X 51.364,Y 103.793,Z 76.328,A 180.000,B 0.000,C 180.000} C_DIS
LIN {X 51.412,Y 103.943,Z 76.323,A 180.000,B 0.000,C 180.000} C_DIS
LIN {X 51.436,Y 104.018,Z 76.320,A 180.000,B 0.000,C 180.000} C_DIS
LIN {X 51.462,Y 104.092,Z 76.317,A 180.000,B 0.000,C 180.000} C_DIS
LIN {X 51.490,Y 104.166,Z 76.314,A 180.000,B 0.000,C 180.000} C_DIS
LIN {X 51.521,Y 104.238,Z 76.312,A 180.000,B 0.000,C 180.000} C_DIS
LIN {X 51.582,Y 104.384,Z 76.306,A 180.000,B 0.000,C 180.000} C_DIS
LIN {X 51.673,Y 104.601,Z 76.298,A 180.000,B 0.000,C 180.000} C_DIS
LIN {X 51.705,Y 104.674,Z 76.295,A 180.000,B 0.000,C 180.000} C_DIS
LIN {X 51.738,Y 104.745,Z 76.292,A 180.000,B 0.000,C 180.000} C_DIS
LIN {X 51.774,Y 104.815,Z 76.290,A 180.000,B 0.000,C 180.000} C_DIS
LIN {X 51.848,Y 104.954,Z 76.284,A 180.000,B 0.000,C 180.000} C_DIS
LIN {X 51.959,Y 105.163,Z 76.276,A 180.000,B 0.000,C 180.000} C_DIS
LIN {X 51.996,Y 105.232,Z 76.273,A 180.000,B 0.000,C 180.000} C_DIS
LIN {X 52.034,Y 105.301,Z 76.270,A 180.000,B 0.000,C 180.000} C_DIS
LIN {X 52.076,Y 105.368,Z 76.268,A 180.000,B 0.000,C 180.000} C_DIS
LIN {X 52.118,Y 105.434,Z 76.265,A 180.000,B 0.000,C 180.000} C_DIS
LIN {X 52.204,Y 105.566,Z 76.259,A 180.000,B 0.000,C 180.000} C_DIS
LIN {X 52.247,Y 105.633,Z 76.257,A 180.000,B 0.000,C 180.000} C_DIS
LIN {X 52.332,Y 105.765,Z 76.251,A 180.000,B 0.000,C 180.000} C_DIS
LIN {X 52.376,Y 105.830,Z 76.248,A 180.000,B 0.000,C 180.000} C_DIS
LIN {X 52.422,Y 105.894,Z 76.246,A 180.000,B 0.000,C 180.000} C_DIS
LIN {X 52.470,Y 105.957,Z 76.243,A 180.000,B 0.000,C 180.000} C_DIS
LIN {X 52.567,Y 106.081,Z 76.237,A 180.000,B 0.000,C 180.000} C_DIS
LIN {X 52.616,Y 106.143,Z 76.235,A 180.000,B 0.000,C 180.000} C_DIS
LIN {X 52.713,Y 106.267,Z 76.229,A 180.000,B 0.000,C 180.000} C_DIS
LIN {X 52.762,Y 106.328,Z 76.226,A 180.000,B 0.000,C 180.000} C_DIS
LIN {X 52.812,Y 106.389,Z 76.224,A 180.000,B 0.000,C 180.000} C_DIS
LIN {X 52.865,Y 106.447,Z 76.221,A 180.000,B 0.000,C 180.000} C_DIS
LIN {X 52.919,Y 106.505,Z 76.218,A 180.000,B 0.000,C 180.000} C_DIS
LIN {X 53.080,Y 106.677,Z 76.210,A 180.000,B 0.000,C 180.000} C_DIS
LIN {X 53.134,Y 106.735,Z 76.207,A 180.000,B 0.000,C 180.000} C_DIS
LIN {X 53.188,Y 106.792,Z 76.204,A 180.000,B 0.000,C 180.000} C_DIS
LIN {X 53.243,Y 106.849,Z 76.202,A 180.000,B 0.000,C 180.000} C_DIS
LIN {X 53.299,Y 106.903,Z 76.199,A 180.000,B 0.000,C 180.000} C_DIS
LIN {X 53.358,Y 106.956,Z 76.196,A 180.000,B 0.000,C 180.000} C_DIS
LIN {X 53.475,Y 107.061,Z 76.191,A 180.000,B 0.000,C 180.000} C_DIS
LIN {X 53.593,Y 107.166,Z 76.185,A 180.000,B 0.000,C 180.000} C_DIS
LIN {X 53.651,Y 107.219,Z 76.182,A 180.000,B 0.000,C 180.000} C_DIS
LIN {X 53.710,Y 107.271,Z 76.180,A 180.000,B 0.000,C 180.000} C_DIS
LIN {X 53.771,Y 107.321,Z 76.177,A 180.000,B 0.000,C 180.000} C_DIS
LIN {X 53.833,Y 107.369,Z 76.174,A 180.000,B 0.000,C 180.000} C_DIS
LIN {X 53.896,Y 107.416,Z 76.172,A 180.000,B 0.000,C 180.000} C_DIS
LIN {X 53.959,Y 107.464,Z 76.169,A 180.000,B 0.000,C 180.000} C_DIS
LIN {X 54.086,Y 107.558,Z 76.164,A 180.000,B 0.000,C 180.000} C_DIS
LIN {X 54.149,Y 107.605,Z 76.161,A 180.000,B 0.000,C 180.000} C_DIS
LIN {X 54.212,Y 107.652,Z 76.159,A 180.000,B 0.000,C 180.000} C_DIS
LIN {X 54.276,Y 107.698,Z 76.156,A 180.000,B 0.000,C 180.000} C_DIS
LIN {X 54.342,Y 107.741,Z 76.154,A 180.000,B 0.000,C 180.000} C_DIS
LIN {X 54.409,Y 107.783,Z 76.151,A 180.000,B 0.000,C 180.000} C_DIS
LIN {X 54.476,Y 107.824,Z 76.149,A 180.000,B 0.000,C 180.000} C_DIS
LIN {X 54.610,Y 107.907,Z 76.144,A 180.000,B 0.000,C 180.000} C_DIS
